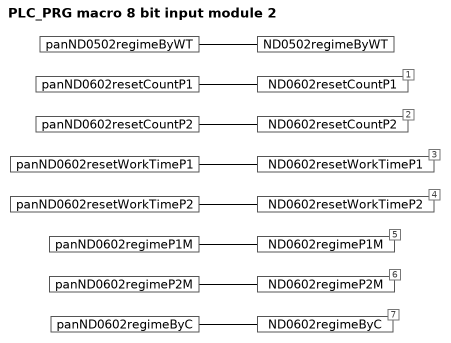
[picture p72: PLC_PRG macro 8 bit input module 2 (CFC)]
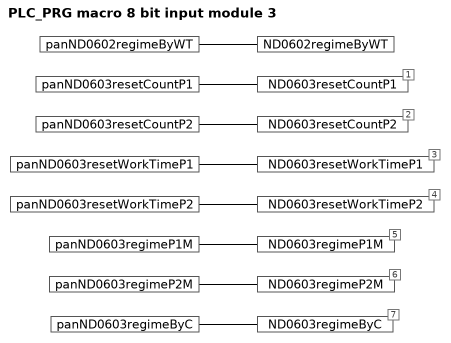
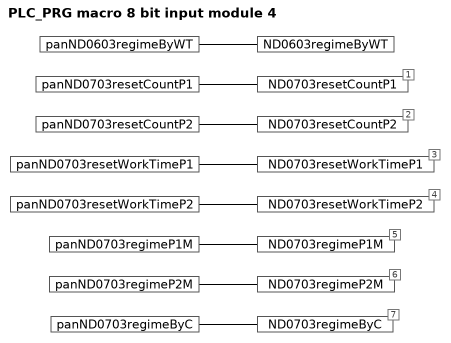
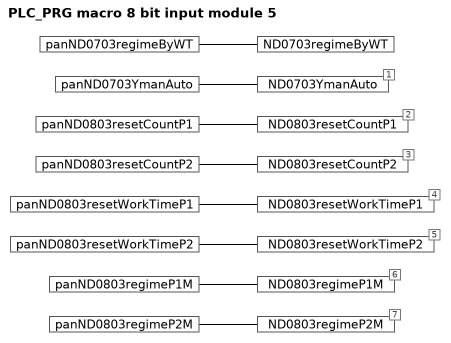
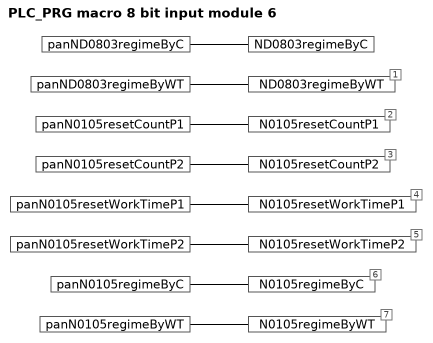
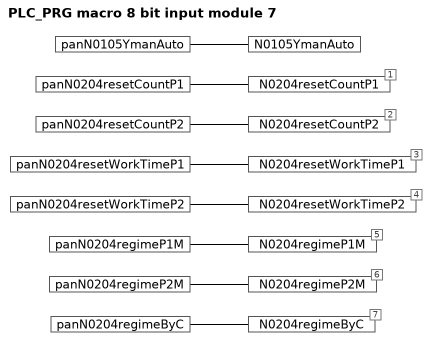
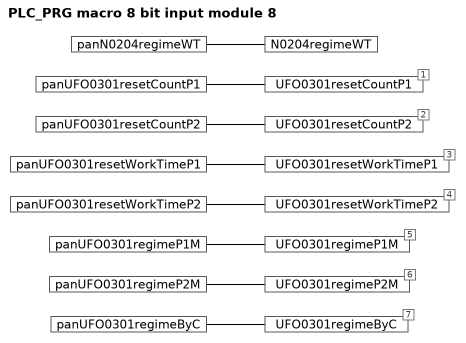
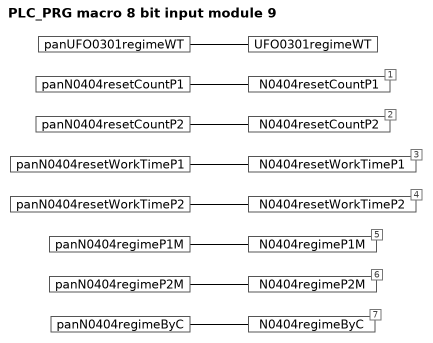
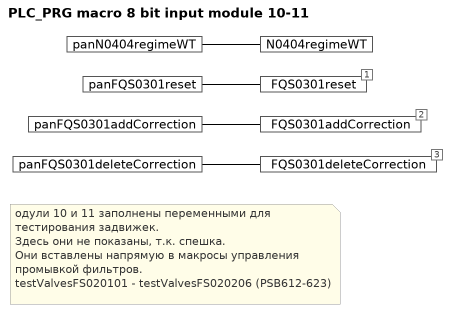
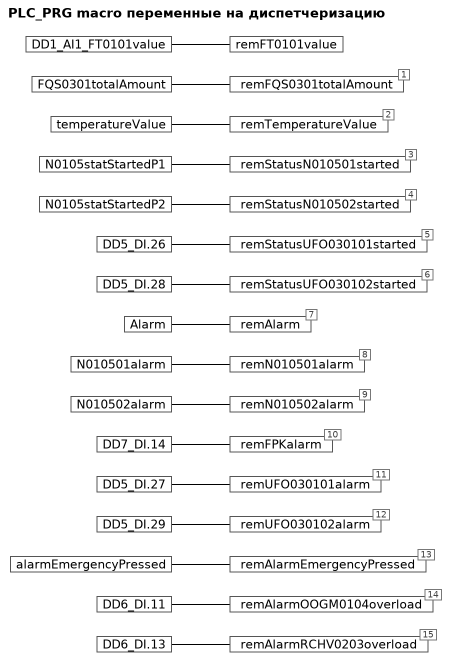
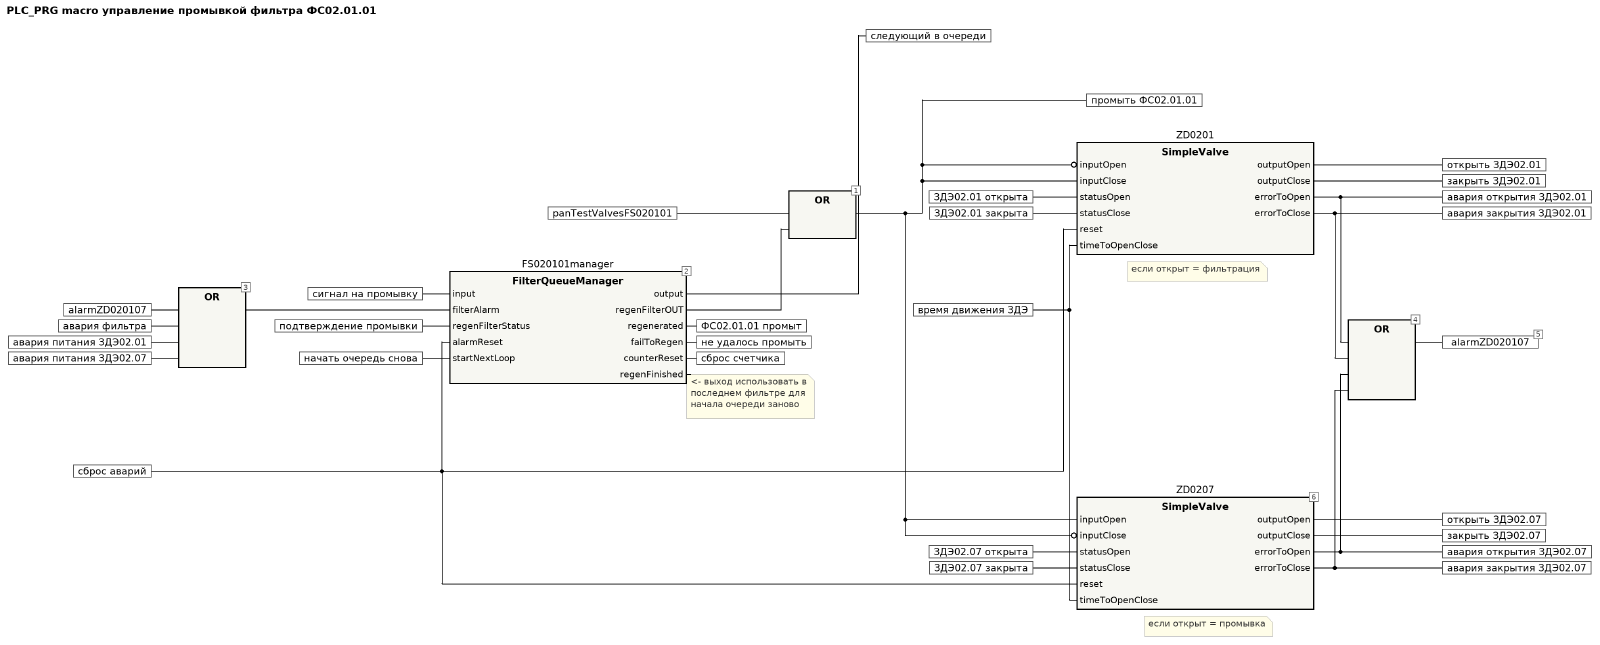
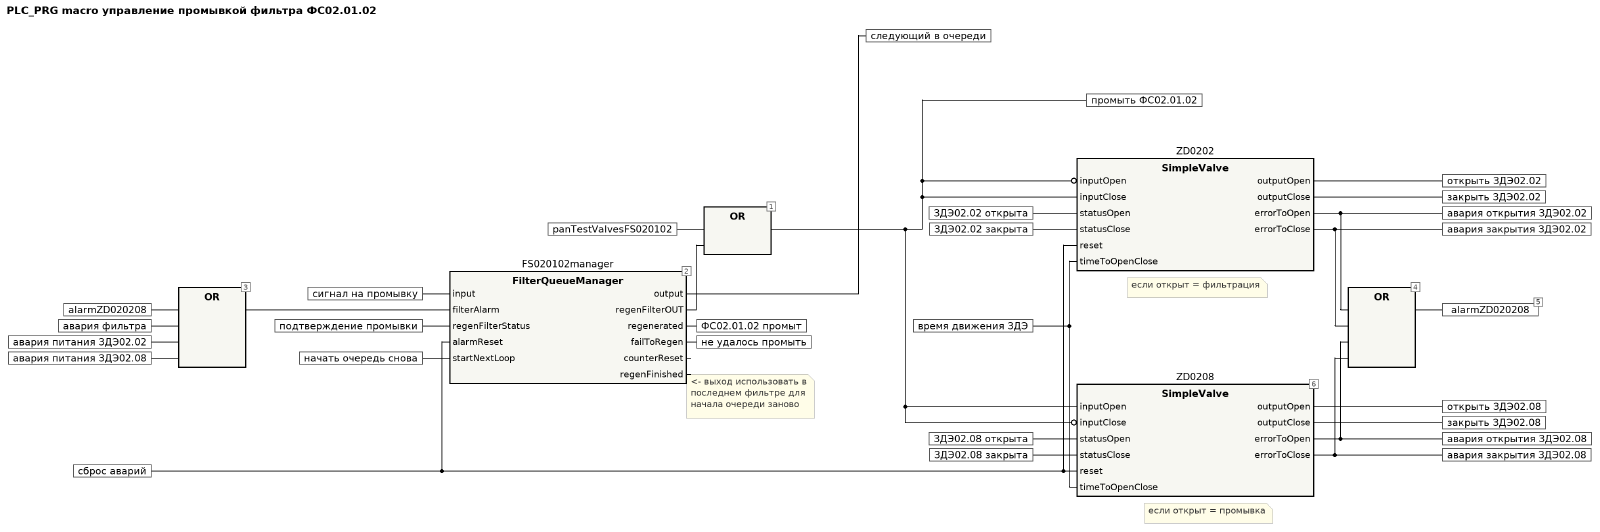
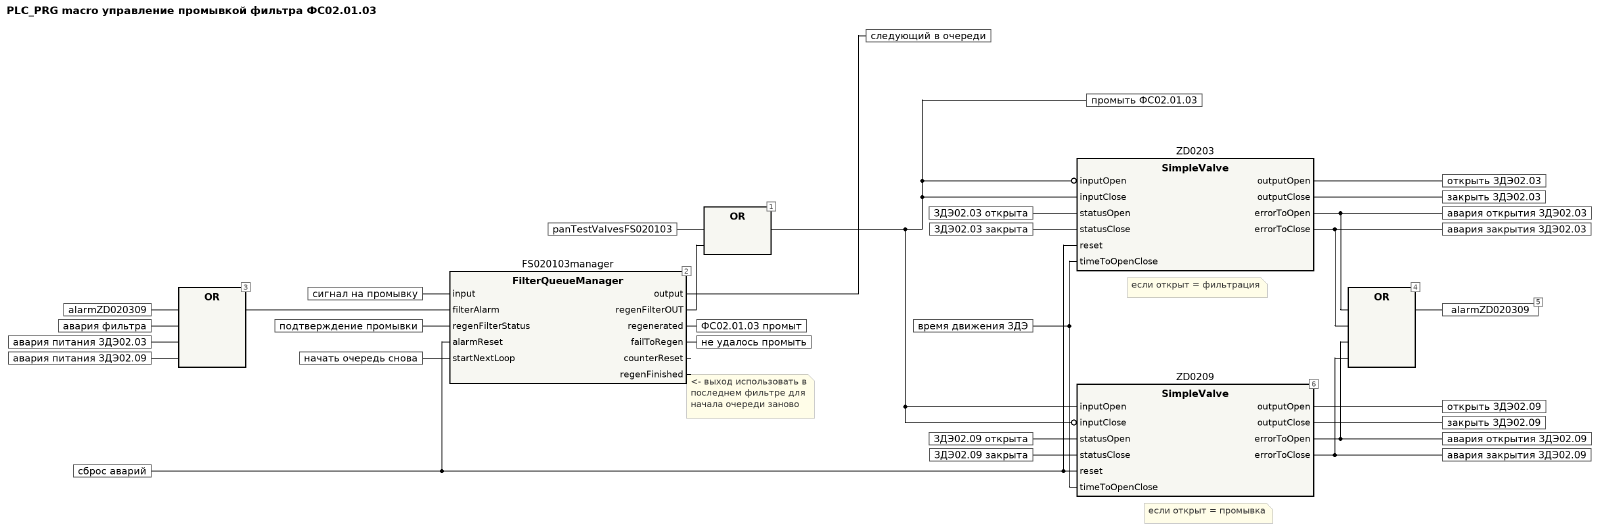
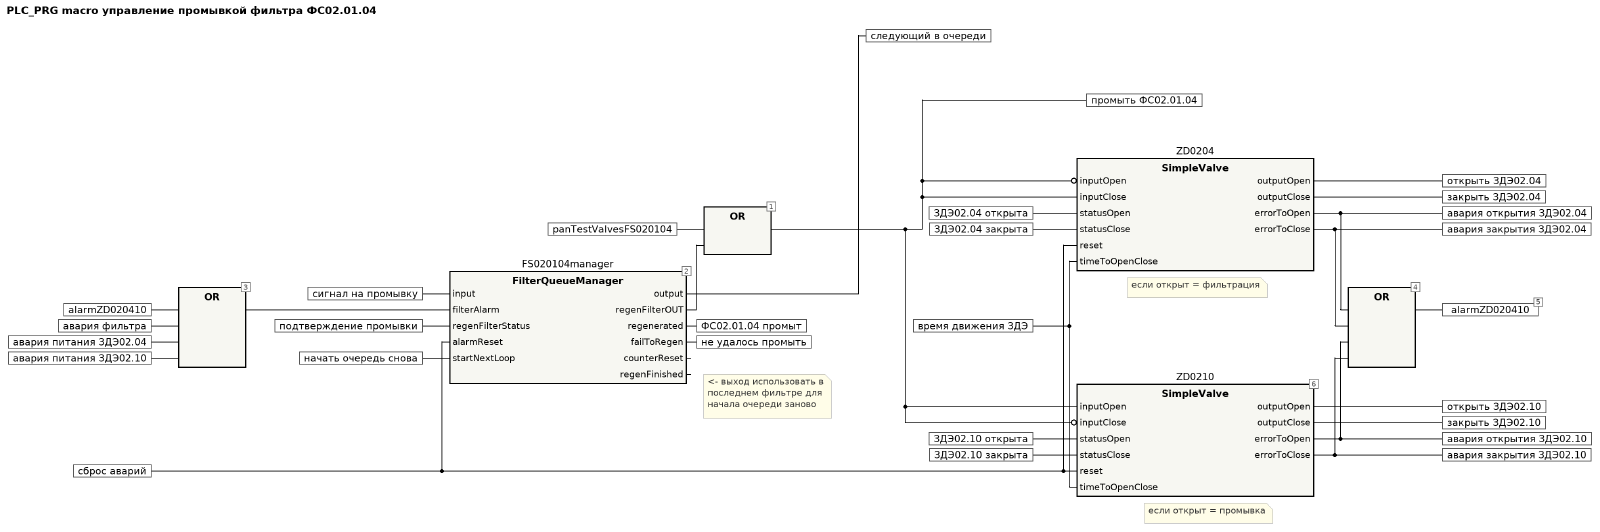
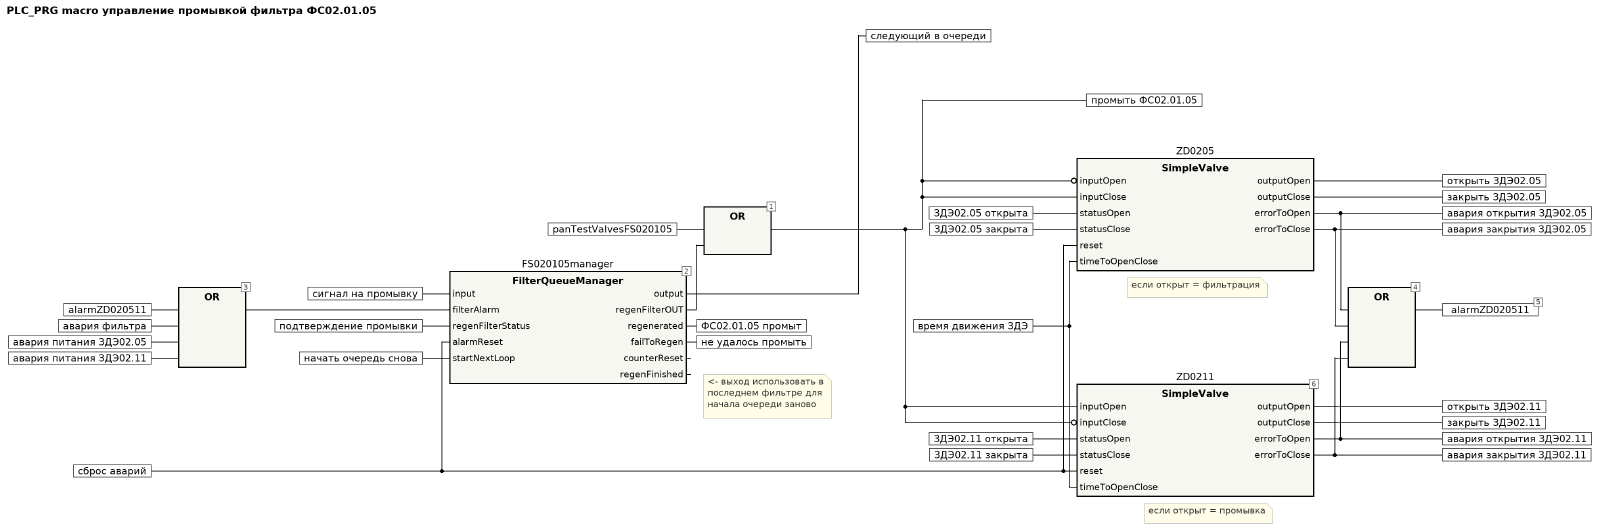
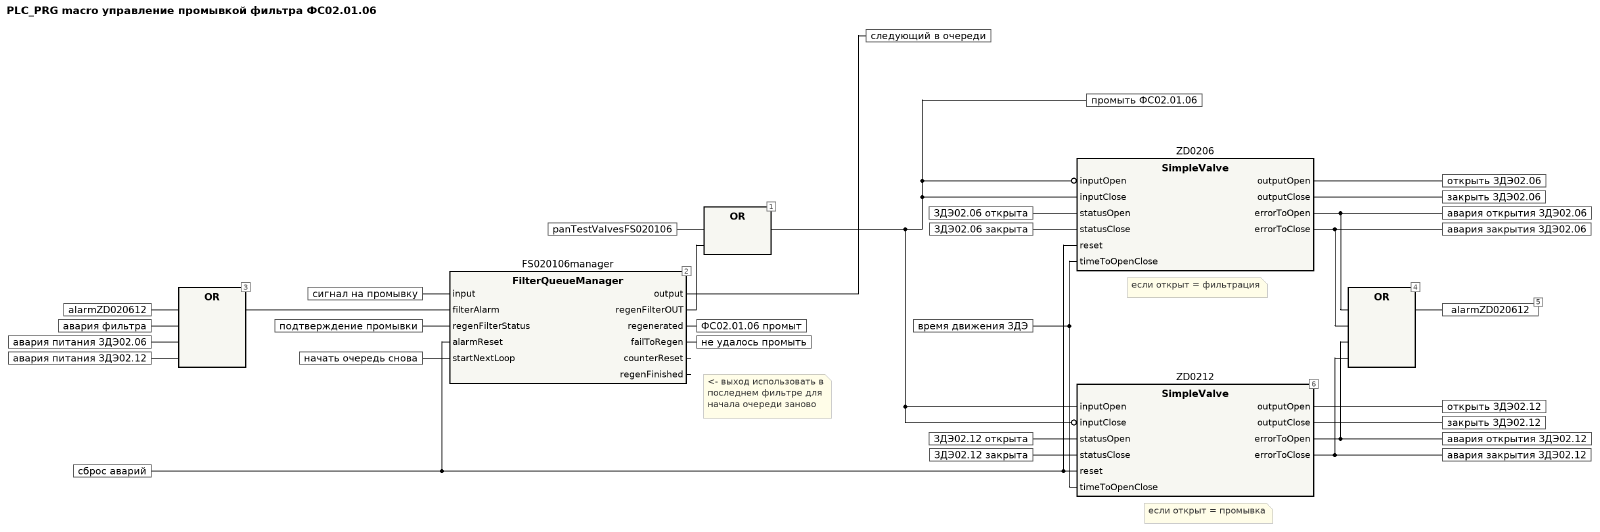
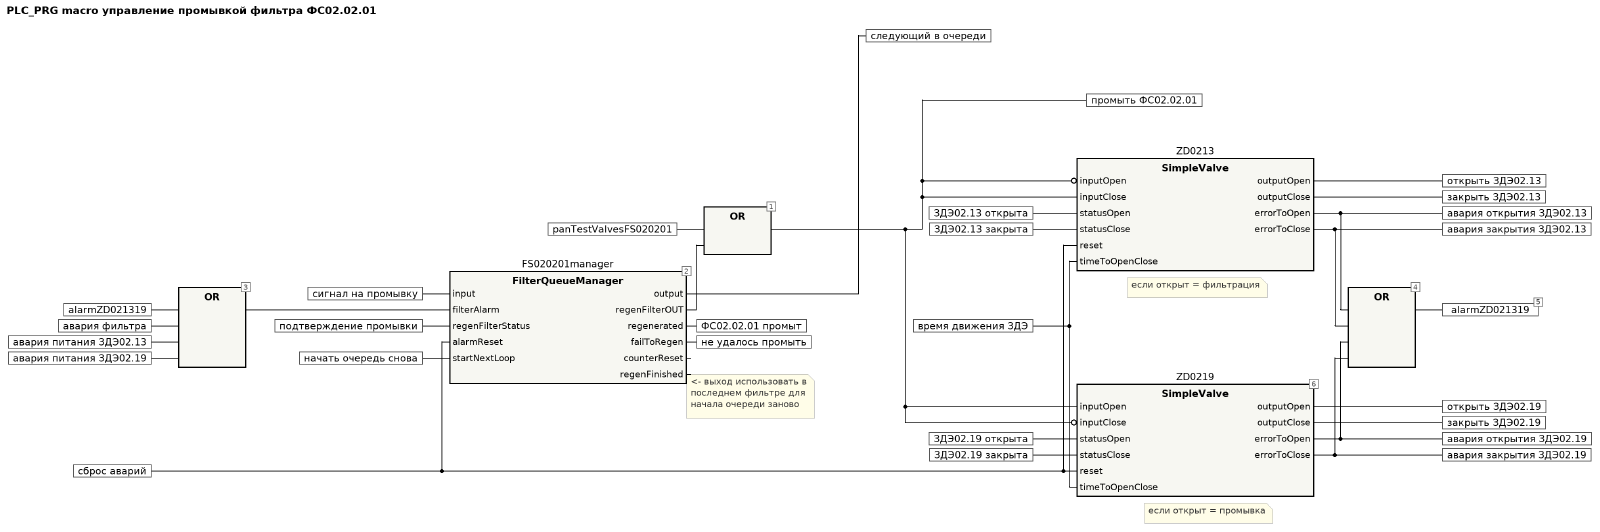
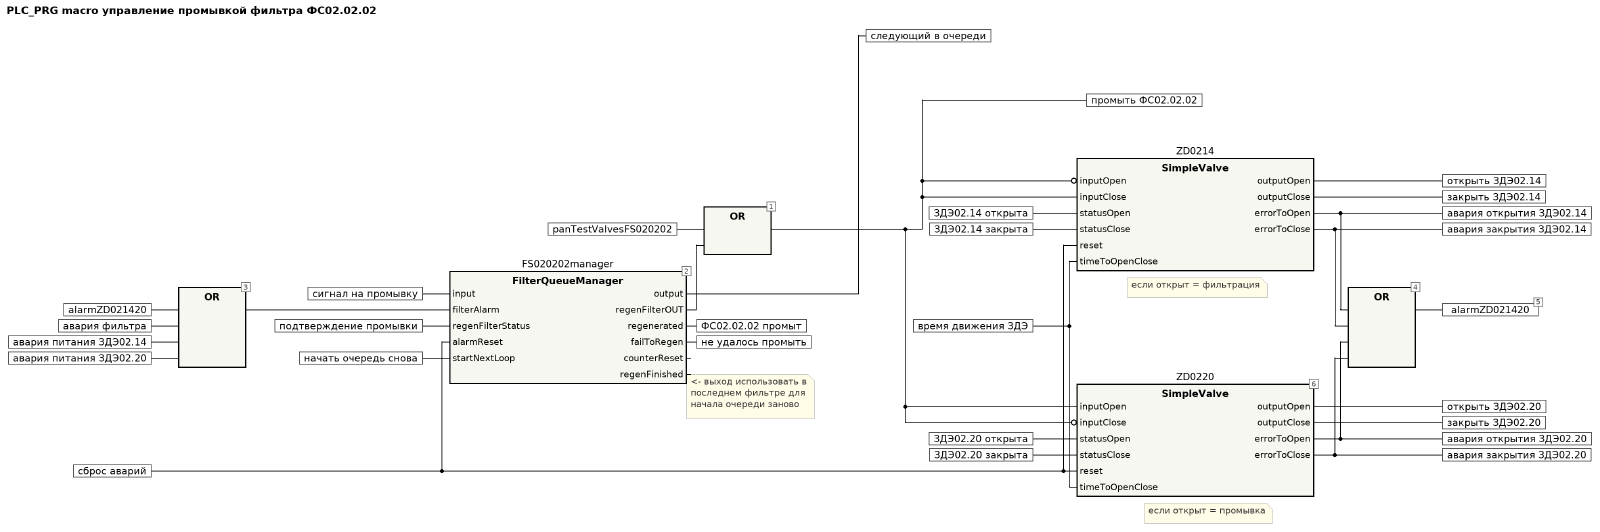
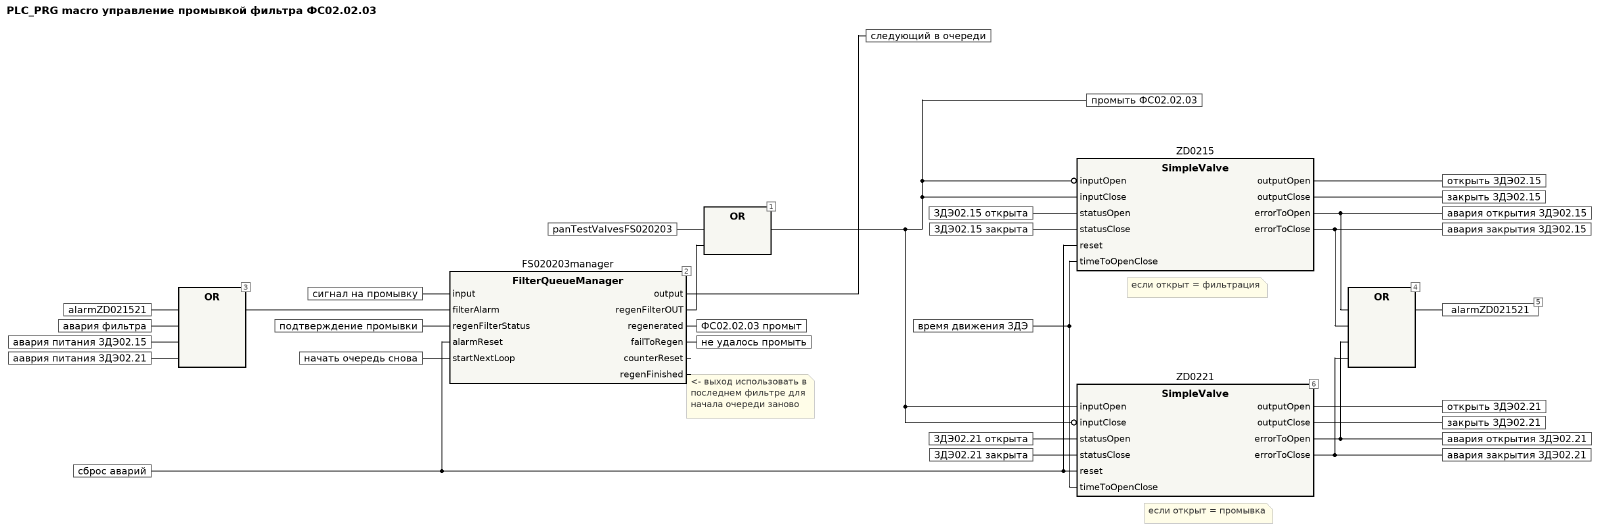
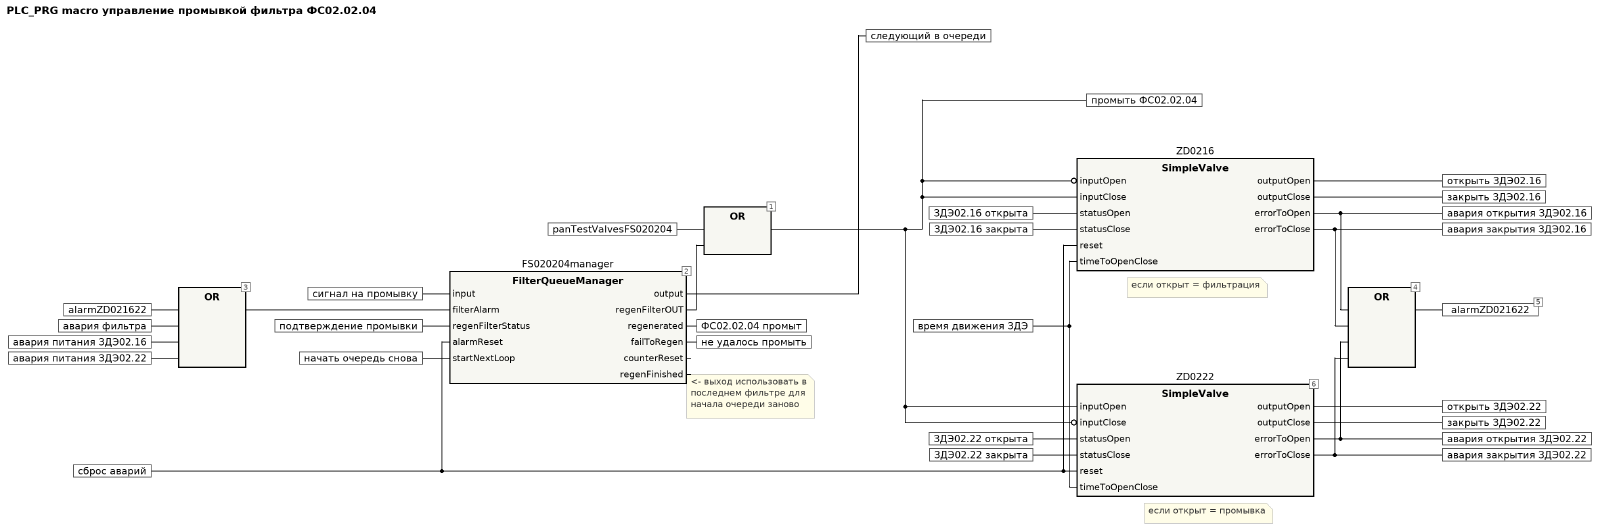
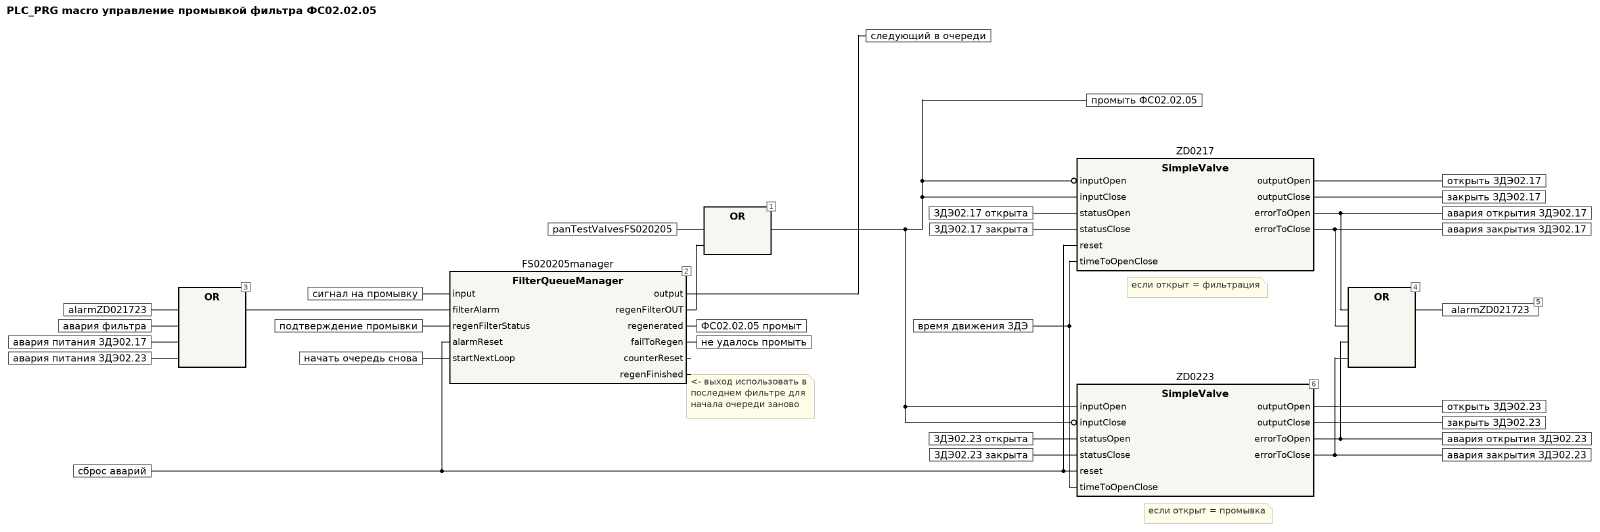
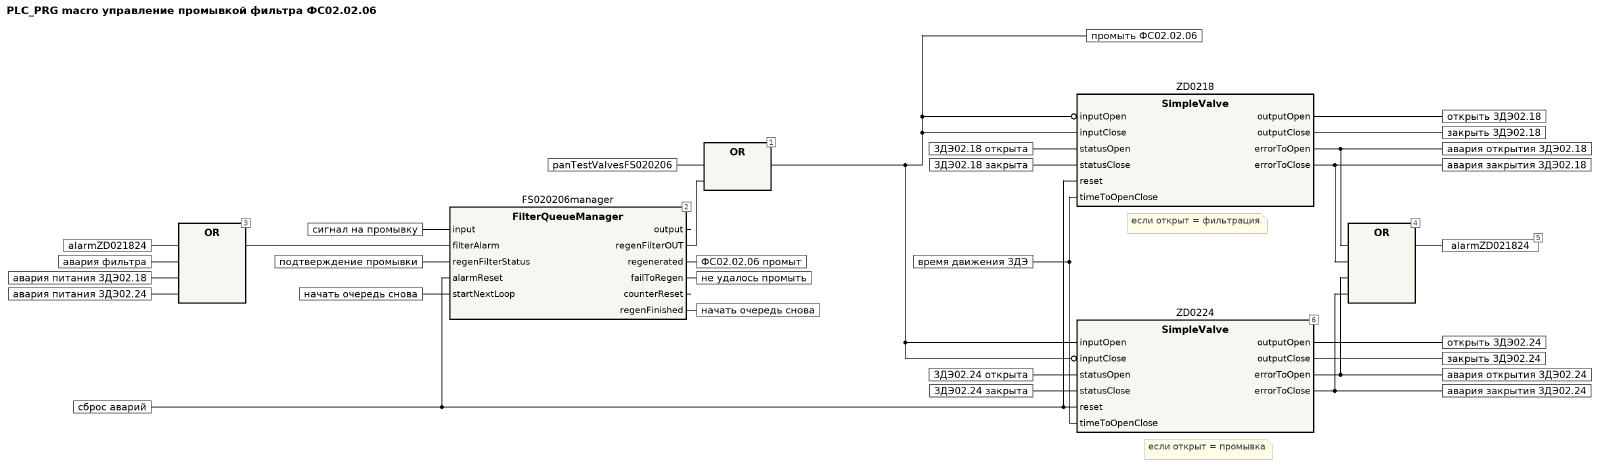
_CFC_ (* Continuous Function Chart, elements in execution order *)
(* 0 = перелив *)
(* авария обоих УФО, если проблемы / открытия/закрытия на одной из задвижек *)
(* авария питания ЗДЭ03.02 *)
(* авария питания ЗДЭ03.01 *)
(* статус-пуск Н01.05/02 *)
(* вкл КМ3 *)
(* Статус ПУСК / ЧРП Н01.05 *)
(* статус-пуск Н01.05/01 *)
(* вкл КМ2 *)
(* контроль обрыва или ошибок модулей в сети ПЛК *)
(* LSA01.02 перелив ОГМ01.04 *)
(* Нажат аварийный стоп. *)
(* авария сети (РКФ) *)
(* разрешение работы КНС / 1 = разрешено *)
(* Нажат аварийный стоп. *)
(* Блок управления разрешением работы КНС *)
(* авария сети (РКФ) *)
(* Авария питания клапанов КЭМ. *)
(* Авария питания розеток / управл.клапанов фильтров. *)
(* авария КНС *)
(* блок подачи сигнала на промывку *)
(* суммируем каждую секунду значение / мгновенного расхода в кубометрах в секунду *)
(* преобразуем расход из / кубометров в час в / кубометры в секунду *)
(* если есть расход / (больше нуля) *)
(* выдает импульс / каждую секунду *)
(* здесь мгновенный расход / в кубометрах в час (FT01.02) *)
(* Авария Н02.04/01 (0=авария) *)
(* Авария Н02.04/02 (0=авария) *)
(* промывка ФС02.01/06 *)
(* промывка ФС02.01/05 *)
(* промывка ФС02.01/04 *)
(* промывка ФС02.01/03 *)
(* промывка ФС02.01/02 *)
(* промывка ФС02.01/01 *)
(* пуск/стоп НД08.03/01 *)
(* пуск/стоп НД08.03/02 *)
(* пуск/стоп НД06.03/01 *)
(* пуск/стоп НД06.03/02 *)
(* пуск/стоп НД06.02/01 *)
(* пуск/стоп НД06.02/02 *)
(* пуск/стоп НД08.04 *)
(* пуск/стоп НД07.03/01 *)
(* пуск/стоп НД07.03/02 *)
(* авария М08.02 (УПФ) *)
(* авария М07.02 (УПЩ) *)
(* авария М06.04 (УПК) *)
(* работа М08.02 (УПФ) *)
(* работа М07.02 (УПЩ) *)
(* работа М06.04 (УПК) *)
(* Контроль, если УФО включили вручную, / а потока при этом нет. *)
(* авария УФО03.01/02 *)
(* работа УФО03.01/02 *)
(* авария УФО03.01/01 *)
(* Для подачи предостережения на пульте / оператора (при необходимости), а также / сигнализации лампой АВАРИЯ. *)
(* работа УФО03.01/01 *)
(* авария УФО03.01/02 *)
(* авария УФО03.01/01 *)
(* авария Н04.04/01 *)
(* авария Н04.04/02 *)
(* время контроля старта ФПК (по умолч.=3мин) *)
(* время работы ФПК после спада сигнала датч.осадка *)
(* запуск фильтрации *)
(* Защита от сухого хода насоса ФПК *)
(* датчик уровня осадка *)
(* Давление на входе ФПК (0...16 бар) *)
(* авария ФПК *)
(* подающий насос ФПК работает *)
(* ФПК готов к приему *)
(* ФПК не запустился *)
(* рН-метр QE01.02 на входе, / диапазон 0...14 *)
(* авария входа рН-метра QE01.01 *)
(* авария входа расходомера FT01.02 *)
(* расходомер FT01.01 на входе, / диапазон 0...600куб/час *)
(* авария НД08.04 *)
(* управление 4...20мА НД08.03/01 *)
(* пуск/стоп НД08.03/01 *)
(* пуск/стоп НД08.03/02 *)
(* управление 4...20мА НД08.03/02 *)
(* авария привода НД08.03/01 *)
(* авария привода НД08.03/02 *)
(* авария НД07.03/01 *)
(* авария НД07.03/02 *)
(* управление 4...20мА НД07.03/01 *)
(* управление 4...20мА НД07.03/02 *)
(* пуск/стоп НД07.03/01 *)
(* пуск/стоп НД07.03/02 *)
(* авария НД07.03/01 *)
(* авария НД07.03/02 *)
(* авария НД06.03/01 *)
(* авария НД06.03/02 *)
(* авария НД06.02/01 *)
(* авария НД06.02/02 *)
(* управление 4...20мА НД06.03/01 *)
(* пуск/стоп НД06.03/01 *)
(* пуск/стоп НД06.03/02 *)
(* управление 4...20мА НД06.03/02 *)
(* авария НД06.03/01 *)
(* авария НД06.03/02 *)
(* управление 4...20мА НД06.02/01 *)
(* пуск/стоп НД06.02/01 *)
(* пуск/стоп НД06.02/02 *)
(* управление 4...20мА НД06.02/02 *)
(* авария НД06.02/01 *)
(* авария НД06.02/02 *)
(* ошибка блока дозирования НД05.02 *)
(* авария входа датчика температуры *)
(* лампа АВАРИЯ *)
(* датчик температуры в помещении / (метран) диапазон: 0...+100С *)
(* управление 4...20мА НД05.02/01 *)
(* пуск/стоп НД05.02/01 *)
(* авария НД05.02/01 *)
(* авария НД05.02/02 *)
(* пуск/стоп НД05.02/02 *)
(* управление 4...20мА НД05.02/02 *)
(* АВАРИИ *)
(* авария привода НД08.03/01 *)
(* авария привода НД08.03/02 *)
(* авария НД08.04 *)
(* насос Н04.01 работает *)
(* пуск/стоп НД08.04 *)
(* управление 4...20мА НД08.04 *)
(* авария входа расходомера FT01.01 *)
(* расходомер FT01.02 на входе, / диапазон 0...600куб/час *)
(* рН-метр QE01.01 на входе, / диапазон 0...14 *)
(* авария входа рН-метра QE01.02 *)
(* сухой ход НД08.03/01 *)
(* сухой ход НД08.03/02 *)
(* сухой ход НД08.03/01 *)
(* сухой ход НД08.03/02 *)
(* LSA01.02 перелив ОГМ01.04 *)
(* Инициализирует требуемые булевые переменные / в момент старта выполнения программы. *)
(* Статус ПУСК ЧРП Н01.05 *)
(* LS01.03 - рабочий верхний уровень ОГМ01.04 автоматический пуск 01.05 *)
(* LS01.04 - нижний уровень ОГМ01.04, сухой ход Н01.05 *)
(* SA1 Ручной выбор Н01.05/01 = главный *)
(* SA1 Ручной выбор Н01.05/02 = главный *)
(* Стоп  Н01.05 (сброс самоподхвата реле) *)
(* время на создание потока *)
(* Пуск  Н01.05 *)
(* КМ1 питание ЧРП *)
(* КМ2 питание насоса 1 *)
(* КМ3 питание насоса 2 *)
(* Авария ЧРП Н01.05 *)
(* термоконтакт Н01.05/01 *)
(* термоконтакт Н01.05/02 *)
(* авария питания ЗДЭ02.25 *)
(* LSА02.01 Перелив РЧВ02.03 *)
(* Давление на входе ФПК / 0...16 бар (мах допуст.10) *)
(* Авария входа AI6 ПЛК, давл.ФПК *)
(* авария ФПК *)
(* Открыть КШЭ04.01 *)
(* статус КШЭ04.01 открыт *)
(* Закрыть КШЭ04.01 *)
(* статус КШЭ04.01 закрыт *)
(* подающий насос ФПК работает *)
(* стоп Н04.04 *)
(* пуск Н04.04/02 *)
(* пуск Н04.04/01 *)
(* авт.пуск Н04.04 *)
(* сухой ход Н04.04, 0=защита *)
(* авария Н04.04/01, 0=авария *)
(* авария Н04.04/02, 0=авария *)
(* импульсный расходомер *)
(* Авария Н02.04/01 (0=авария) *)
(* Авария Н02.04/02 (0=авария) *)
(* промывка ФС02.02/06 *)
(* промывка ФС02.02/05 *)
(* промывка ФС02.02/04 *)
(* промывка ФС02.02/03 *)
(* промывка ФС02.02/02 *)
(* промывка ФС02.02/01 *)
(* Клапан КЭМ05.01 открыт. *)
(* Клапан КЭМ06.01 открыт. *)
(* Клапан КЭМ07.01 открыт. *)
(* Клапан КЭМ08.01 открыт. *)
(* Сухой ход Н02.04 (LS02.03) 0=сух.ход *)
(* Стоп Н02.04 *)
(* Пуск Н02.04/01 *)
(* Пуск Н02.04/02 *)
(* текущий объем *)
(* заданный до промывки объем *)
(* 0=авария *)
(* авария (при 0) ФС02.01/06 *)
(* авария (при 0) ФС02.01/05 *)
(* авария (при 0) ФС02.01/04 *)
(* авария (при 0) ФС02.01/03 *)
(* авария (при 0) ФС02.01/02 *)
(* авария (при 0) ФС02.01/01 *)
(* авария (при 0) ФС02.02/06 *)
(* авария (при 0) ФС02.02/05 *)
(* авария (при 0) ФС02.02/04 *)
(* авария (при 0) ФС02.02/03 *)
(* авария (при 0) ФС02.02/02 *)
(* авария (при 0) ФС02.02/01 *)
(* сброс счетчика стоков до следующей промывки *)
(* подсчет общего объема стоков, прошедшего через расходомер FT01.02 *)
(* очередь передается на 2 ступень *)
(* авария питания ЗДЭ02.01 *)
(* авария питания ЗДЭ02.02 *)
(* авария питания ЗДЭ02.03 *)
(* авария питания ЗДЭ02.04 *)
(* авария питания ЗДЭ02.05 *)
(* авария питания ЗДЭ02.06 *)
(* авария питания ЗДЭ02.07 *)
(* авария питания ЗДЭ02.08 *)
(* авария питания ЗДЭ02.09 *)
(* авария питания ЗДЭ02.10 *)
(* авария питания ЗДЭ02.11 *)
(* авария питания ЗДЭ02.12 *)
(* авария питания ЗДЭ02.13 *)
(* авария питания ЗДЭ02.14 *)
(* авария питания ЗДЭ02.15 *)
(* авария питания ЗДЭ02.16 *)
(* авария питания ЗДЭ02.17 *)
(* авария питания ЗДЭ02.18 *)
(* авария питания ЗДЭ02.19 *)
(* авария питания ЗДЭ02.20 *)
(* авария питания ЗДЭ02.21 *)
(* авария питания ЗДЭ02.22 *)
(* авария питания ЗДЭ02.23 *)
(* авария питания ЗДЭ02.24 *)
(* инвертирование сигнала, чтобы все аварии / обозначались как 1 (TRUE) *)
(* авария НД05.02/01 *)
(* авария НД05.02/02 *)
(* авария питания КШЭ04.01 *)
(* 1=открыть; 0 = закрыть *)
(* в этом макросе лежит управление режимом тестирования задвижек ЗДЭ03 / Тестирование запрещает автоматический запуск УФО от ПЛК *)
#0 rTrigStartInitializer:R_TRIG(CLK: TRUE)
#1 startInitializer <= #0.Q
#2 MACRO контроль температуры в помещении(pin 1 "вход датчика температуры": DD1_AI0, pin 2 "минимально допустимая температура в помещении": maxTemperature, pin 3 "максимально допустимая температура в помещении": minTemperature)
	(* задаем границы допустимой температуры в помещении / проверяем что измеренное значение в заданном диапазоне *)
	(* не смотрим конкретный тип ошибки / (работает не точно, обрыв определяет как слишком маленькое значение) / если не равно 0 - значит на входе ошибка *)
	#3 DD1_AI0_temperature:DECODE_FLOAT(VALUE: pin 1, DEF_VALUE: -)
	#4 NE(#3._ERR, 0)
	out 2 "авария датчика температуры" <= #4
	out 1 "температура в помещении" <= #3.OUT_VALUE
	#5 REAL_TO_INT(#3.OUT_VALUE)
	#6 temperatureLimits:LIMITALARM(IN: #5, HIGH: pin 3, LOW: pin 2)
	out 3 "температура выше заданного диапазона" <= #6.O
	out 4 "температура ниже заданного диапазона" <= #6.U
	#7 temperatureLimits:LIMITALARM(IN: -, HIGH: -, LOW: -)
END_MACRO
#8 temperatureValue <= #2.out 1
#9 DD1_AI0_error <= #2.out 2
#10 alarmHighTemperature <= #2.out 3
#11 alarmLowTemperature <= #2.out 4
#12 OR(testKSHE0401, DD7_DI.13)
#13 MACRO клапан шаровый перед ФПК (КШЭ04.01)(pin 1 "сигнал "подающий насос ФПК" работает": #12, pin 2 "статус КШЭ04.01 открыт": DD9_DI.2, pin 3 "статус КШЭ04.01 закрыт": DD9_DI.3, pin 4 "сброс аварий": alarmReset, pin 5 "время на открытие/закрытие": timeToOpenCloseValve)
	#14 FPKkshe0401DelayToOpen:TON(IN: #16.outputOpen, PT: T#1s)
	out 1 "выход на открытие КШЭ04.01" <= #14.Q
	#15 FPKkshe0401DelayToClose:TON(IN: #16.outputClose, PT: T#1s)
	out 2 "выход на закрытие КШЭ04.01" <= #15.Q
	#16 FPKkshe0401:SimpleValve(inputOpen: pin 1, inputClose: #17, statusOpen: pin 2, statusClose: pin 3, reset: pin 4, timeToOpenClose: pin 5)
	#17 NOT(pin 1)
	out 3 "авария на открытие КШЭ04.01" <= #16.errorToOpen
	out 4 "авария на закрытие КШЭ04.01" <= #16.errorToClose
END_MACRO
#18 DD4_DO.2 <= #13.out 1
#19 DD4_DO.3 <= #13.out 2
#20 FPKkshe0401errorToOpen <= #13.out 3
#21 FPKkshe0401errorToClose <= #13.out 4
#22 OR(DD1_AI0_error, DD1_AI1_error, DD1_AI2_error, DD1_AI3_error, DD1_AI4_error, alarmHighTemperature, alarmLowTemperature, ND0502dosingError, ND0602dosingError, ND0603dosingError, ND0803dosingError, ND0804dosingError, DD1_DI6, DD1_DI7, N010501alarm, N010502alarm, ZDE0225errorToOpen, ZDE0225errorToClose, DD7_DI.14, FPKnotStarted, DD1_AI5_error, FPKkshe0401errorToOpen, FPKkshe0401errorToClose, DD5_DI.27, DD5_DI.29, filterFailToRegen020101, errorToOpenZD0201, errorToCloseZD0201, errorToOpenZD0207, errorToCloseZD0207, filterFailToRegen020102, errorToOpenZD0202, errorToCloseZD0202, errorToOpenZD0208, errorToCloseZD0208, filterFailToRegen020103, errorToOpenZD0203, errorToCloseZD0203, errorToOpenZD0209, errorToCloseZD0209, filterFailToRegen020104, errorToOpenZD0204, errorToCloseZD0204, errorToOpenZD0210, errorToCloseZD0210, filterFailToRegen020105, errorToOpenZD0205, errorToCloseZD0205, errorToOpenZD0211, errorToCloseZD0211, filterFailToRegen020106, errorToOpenZD0206, errorToCloseZD0206, errorToOpenZD0212, errorToCloseZD0212, filterFailToRegen020201, errorToOpenZD0213, errorToCloseZD0213, errorToOpenZD0219, errorToCloseZD0219, filterFailToRegen020202, errorToOpenZD0214, errorToCloseZD0214, errorToOpenZD0220, errorToCloseZD0220, filterFailToRegen020203, errorToOpenZD0215, errorToCloseZD0215, errorToOpenZD0221, errorToCloseZD0221, filterFailToRegen020204, errorToOpenZD0216, errorToCloseZD0216, errorToOpenZD0222, errorToCloseZD0222, filterFailToRegen020205, errorToOpenZD0217, errorToCloseZD0217, errorToOpenZD0223, errorToCloseZD0223, filterFailToRegen020206, errorToOpenZD0218, errorToCloseZD0218, errorToOpenZD0224, errorToCloseZD0224, alarmPLKnetwork, alarmND050201, alarmND050202, alarmND060201, alarmND060202, alarmND060301, alarmND060302, alarmND070301, alarmND070302, alarmND080301, alarmND080302, alarmND0804, alarmOGM0104overload, alarmRCHV0203overload, alarmN040402, alarmN040401, alarmM0604, alarmM0702, alarmM0802, alarmN020401, alarmN020402, alarmFS020101, alarmFS020102, alarmFS020103, alarmFS020104, alarmFS020105, alarmFS020106, alarmFS020201, alarmFS020202, alarmFS020203, alarmFS020204, alarmFS020205, alarmFS020206, alarmZDE0201power, alarmZDE0202power, alarmZDE0203power, alarmZDE0204power, alarmZDE0205power, alarmZDE0206power, alarmZDE0207power, alarmZDE0208power, alarmZDE0209power, alarmZDE0210power, alarmZDE0211power, alarmZDE0212power, alarmZDE0213power, alarmZDE0214power, alarmZDE0215power, alarmZDE0216power, alarmZDE0217power, alarmZDE0218power, alarmZDE0219power, alarmZDE0220power, alarmZDE0221power, alarmZDE0222power, alarmZDE0223power, alarmZDE0224power, alarmZDE0225power, alarmKSHE0401power, alarmKNS, alarmPowerSocketFS, alarmKEMvalvesPower, alarmEmergencyPressed, alarmRKF, errorToOpenZDE0301, errorToCloseZDE0301, errorToOpenZDE0302, errorToCloseZDE0302, alarmZDE0301power, alarmZDE0302power)
#23 DD1_DO11 <= #22
#24 alarm <= #22
#25 MACRO контроль аналогового входа DD1_AI1(pin 1 "вход": DD1_AI1)
	(* Не смотрим конкретную ошибку, / определяем,что вход неисправен без расшифровки. *)
	#26 DD1_AI1_FT0101:DECODE_FLOAT(VALUE: pin 1, DEF_VALUE: -)
	#27 NE(#26._ERR, 0)
	out 2 "авария" <= #27
	out 1 "выход" <= #26.OUT_VALUE
END_MACRO
#28 DD1_AI1_FT0101value <= #25.out 1
#29 DD1_AI1_error <= #25.out 2
#30 MACRO контроль аналогового входа DD1_AI2(pin 1 "вход": DD1_AI2)
	(* Не смотрим конкретную ошибку, / определяем,что вход неисправен без расшифровки. *)
	#31 DD1_AI2_FT0102:DECODE_FLOAT(VALUE: pin 1, DEF_VALUE: -)
	#32 NE(#31._ERR, 0)
	out 2 "авария" <= #32
	out 1 "выход" <= #31.OUT_VALUE
END_MACRO
#33 DD1_AI2_FT0102value <= #30.out 1
#34 DD1_AI2_error <= #30.out 2
#35 MACRO управление Н01.05 (поддержание заданного расхода по FT01.02)(pin 1 "статус ПУСК ЧРП (реле)": DD5_DI.4, pin 2 "LS01.03 раб.уров.": DD6_DI.12, pin 3 "LS01.04 ниж.уров.(сух.ход)": DD5_DI.0, pin 4 "SA1ручной выб.Н01.05/01-главный": DD5_DI.5, pin 5 "SA1ручной выб.Н01.05/02-главный": DD5_DI.6, pin 6 "включить режим "по кол.вкл."": N0105regimeByC, pin 7 "включить режим "по наработке"": N0105regimeByWT, pin 8 "значение расхода от FT01.02": DD1_AI2_FT0102value, pin 9 "уставка расхода": N0105flowSetValue, pin 10 "время на создание потока": N0105minFlowTime, pin 11 "Р-коэфф.": N0105koeffP, pin 12 "I-коэфф": N0105koeffI, pin 13 "Д-коэфф": N0105koeffD, pin 14 "управление ЧРП в ручн.реж.(4...20мА)": N0105YoutManual, pin 15 "переключатель управление ЧРП РУЧН/АВТ": N0105YmanAuto, pin 16 "мин.допустимый расход": N0105minFlow, pin 17 "термоконтакт Н01.05/01": DD5_DI.2, pin 18 "термоконтакт Н01.05/02": DD5_DI.3, pin 19 "авария ЧРП Н01.05": DD5_DI.1, pin 20 "сброс аварии": alarmReset, pin 21 "сброс кол-ва вкл.Н01.05/01": N0105resetCountP1, pin 22 "сброс кол-ва вкл.Н01.05/02": N0105resetCountP2, pin 23 "сброс наработки Н01.05/01": N0105resetWorkTimeP1, pin 24 "сброс наработки Н01.05/02": N0105resetWorkTimeP2)
	(* время на создание потока *)
	(* Пуск  Н01.05 *)
	(* режимы по количеству включений,  или по наработке / активны если оба входа SA1 не активны *)
	(* управление Н01.05 - поддержание / заданного расхода по FT01.02 *)
	(* по умолчанию при старте программы *)
	(* если на входе true / то нижнее значение, / иначе то, что посередине *)
	(* Если насос создает давление меньше / указанного, то авария. *)
	#36 OR(pin 2, #37.Q)
	#37 N0105startTrig:R_TRIG(CLK: pin 1)
	#38 N0105stopTrig:F_TRIG(CLK: pin 1)
	#39 N0105startTrigg:RS(SET: #36, RESET1: #41)
	#40 N0105regime:choosePumpRegime(start: #39.Q1, pump1Main: pin 4, pump2Main: pin 5, byCounter: #44, byWorkTime: #50)
	out 2 "статус режим "Н01.05/01 - главный"" <= #40.pump1MainActive
	out 3 "статус режим "Н01.05/02 - главный"" <= #40.pump2MainActive
	out 4 "статус режим "по кол-ву вкл."" <= #40.byCounterActive
	#41 OR(#38.Q, #42)
	out 5 "статус режим "по наработке"." <= #40.byWorkTimeActive
	#42 NOT(pin 3)
	#43 NOT(#39.Q1)
	out 1 "СТОП (сброс самоподхвата реле пуска ЧРП)." <= #43
	#44 AND(NOT pin 4, NOT pin 5, #47.Q1)
	#45 OR(pin 6, startInitializer)
	#46 N0105regByCinit:R_TRIG(CLK: #45)
	#47 N0105regByCtrig:RS(SET: #46.Q, RESET1: #55.Q)
	#48 N0105twoPumpOneDriveManager:TwoPumpOneDriveManager(startStopPump1: #40.startPump1, startStopPump2: #40.startPump2, alarmPump1: N010501alarm, alarmPump2: N010502alarm, alarmReset: alarmReset, counterStart: #40.startByCounter, Pump1ResetCounter: pin 21, Pump2ResetCounter: pin 22, ValueToResetCounter: -, workTimeStart: #40.startByWorkTime, workTimePump1Reset: pin 23, workTimePump2Reset: pin 24, timeKM1off: -, timeKM23DelayON: -, timeKM23offDelay: -, timeReadyToStartDelay: -)
	out 6 "кол-во включений Н01.05/01" <= #48.counterPump1
	#49 AND(#48.pump1active, #65)
	out 7 "кол-во включений Н01.05/02" <= #48.counterPump2
	out 8 "наработка Н01.05/01" <= #48.currentWorkTimePump1
	out 15 "авария Н01.05/01" <= #53.Q1
	#50 AND(NOT pin 4, NOT pin 5, #56.Q1)
	out 9 "наработка Н01.05/02" <= #48.currentWorkTimePump2
	out 10 "КМ1-питание ЧРП" <= #48.DriveKM
	#51 AND(#48.pump1active, #57)
	#52 OR(#49, #51)
	#53 N010501alarmTrig:RS(SET: #52, RESET1: pin 20)
	#54 N010501alarm <= #53.Q1
	#55 N0105regWTinit:R_TRIG(CLK: pin 7)
	#56 N0105regWTtrig:RS(SET: #55.Q, RESET1: #46.Q)
	out 11 "КМ2-питание Н01.05/01" <= #48.pump1KM
	out 12 "КМ3-питание Н01.05/02" <= #48.pump2KM
	#57 OR(NOT pin 17, NOT pin 19)
	out 13 "пуск ЧРП (Н01.05)" <= #48.driveStart
	#58 OR(NOT pin 19, NOT pin 18)
	out 16 "авария Н01.05/02" <= #61.Q1
	#59 AND(#58, #48.pump2active)
	#60 OR(#59, #63)
	#61 N010502alarmTrig:RS(SET: #60, RESET1: pin 20)
	#62 N010502alarm <= #61.Q1
	#63 AND(#48.pump2active, #65)
	#64 N0105timerminFlow:TON(IN: #48.driveStart, PT: pin 10)
	#65 AND(#64.Q, #66)
	#66 LE(pin 8, pin 16)
	#67 SEL(#48.driveStart, 0, #68.Y)
	out 14 "управление ЧРП (4...20мА)" <= #67
	#68 N0105pidReg:PID(ACTUAL: pin 8, SET_POINT: pin 9, KP: pin 11, TN: pin 12, TV: pin 13, Y_MANUAL: pin 14, Y_OFFSET: -, Y_MIN: 4, Y_MAX: 20, MANUAL: pin 15, RESET: #68.OVERFLOW)
END_MACRO
#69 DD4_DO.13 <= #35.out 1
#70 N0105statRegimeP1M <= #35.out 2
#71 N0105statRegimeP2M <= #35.out 3
#72 N0105statRegimeByC <= #35.out 4
#73 N0105statRegimeByWT <= #35.out 5
#74 N0105counterP1 <= #35.out 6
#75 N0105counterP2 <= #35.out 7
#76 N0105workTimeP1 <= #35.out 8
#77 N0105workTimeP2 <= #35.out 9
#78 DD2_DO.0 <= #35.out 10
#79 DD2_DO.1 <= #35.out 11
#80 DD2_DO.2 <= #35.out 12
#81 DD1_DO0 <= #35.out 13
#82 DD1_AO0 <= #35.out 14
#83 N010501alarm <= #35.out 15
#84 N010502alarm <= #35.out 16
#85 MACRO Сигналы работы с ФП04.02 (фильтр-пресс)(pin 1 "датчик уровня осадка": DD7_DI.15, pin 2 "время работы ФПК (после выкл.датч.осадка)": FPKtimeToWork, pin 3 "защита от сухого хода": DD6_DI.10, pin 4 "ошибка входа AI (обрыв)": DD1_AI5_error, pin 5 "авария ФПК": DD7_DI.14, pin 6 "фильтр-пресс готов к приему": DD7_DI.12, pin 7 "давление на входе в ФПК": DD1_AI5_FPKpressureValue, pin 8 "мах допустимое давление": FPKmaxPressureValue, pin 9 "подающий насос ФПК работает": DD7_DI.13, pin 10 "время контроля старта ФПК": FPKnotStartedTime, pin 11 "сброс аварий": alarmReset)
	(* ФПК готов к приему осадка *)
	(* LS01.01-нижн.уровень на входе ОГМ01.04 / защита от сух. хода насоса ФПК *)
	(* LES01.01-сигнал датчика уровня осадка ОГМ01.04 / запуск процесса фильтрации *)
	(* Время работы ФПК после / спада сигнала уровня осадка / по умолч.15мин. *)
	(* Давление на входе ФПК / 0...16 бар (мах допуст.10) *)
	(* максимально допустимое давление / на входе ФПК *)
	(* Условие сброса сигнала о грязном фильтр-прессе: / 1. Пропал сигнал о готовности ФПК; / 2. Появился сигнал о готовности ФПК. / Это значит, что оператор раздвигал плиты, / чистил и снова сдвигал их. *)
	#86 FPKneedToCleanResetFtrig:F_TRIG(CLK: FPKneedToCleanReset)
	#87 FPKstartTrig:RS(SET: pin 1, RESET1: #93)
	out 1 "запуск/старт ФПК" <= #87.Q1
	#88 FPKstopTimer:TOF(IN: pin 1, PT: pin 2)
	#89 FPKstopFtrig:F_TRIG(CLK: #88.Q)
	#90 AND(#87.Q1, #91)
	#91 NOT(pin 11)
	#92 AND(#87.Q1, #94.Q, #96)
	out 2 "ФПК не стартовал" <= #92
	#93 OR(#89.Q, pin 4, pin 5, #95, #97, #100.Q1)
	#94 FPKnotStartedTimer:TON(IN: #90, PT: pin 10)
	#95 NOT(pin 3)
	#96 NOT(pin 9)
	#97 NOT(pin 6)
	#98 AND(#87.Q1, #99)
	#99 GE(pin 7, pin 8)
	#100 FPKneedToCleanTrig:RS(SET: #98, RESET1: #86.Q)
	out 3 "ФПК нужно почистить!" <= #100.Q1
	#101 S FPKneedToCleanReset <= #100.Q1
	#102 FPKneedToCleanResetRtrig:R_TRIG(CLK: pin 6)
	#103 R FPKneedToCleanReset <= #102.Q
END_MACRO
#104 DD1_DO10 <= #85.out 1
#105 FPKnotStarted <= #85.out 2
#106 FPKneedToClean <= #85.out 3
#107 MACRO контроль аналогового входа DD1_AI3(pin 1 "вход": DD1_AI3)
	(* Не смотрим конкретную ошибку, / определяем,что вход неисправен без расшифровки. *)
	#108 DD1_AI3_QE0101:DECODE_FLOAT(VALUE: pin 1, DEF_VALUE: -)
	#109 NE(#108._ERR, 0)
	out 2 "авария" <= #109
	out 1 "выход" <= #108.OUT_VALUE
END_MACRO
#110 DD1_AI3_QE0101value <= #107.out 1
#111 DD1_AI3_error <= #107.out 2
#112 MACRO контроль аналогового входа DD1_AI4(pin 1 "вход": DD1_AI4)
	(* Не смотрим конкретную ошибку, / определяем,что вход неисправен без расшифровки. *)
	#113 DD1_AI4_QE0102:DECODE_FLOAT(VALUE: pin 1, DEF_VALUE: -)
	#114 NE(#113._ERR, 0)
	out 2 "авария" <= #114
	out 1 "выход" <= #113.OUT_VALUE
END_MACRO
#115 DD1_AI4_QE0102value <= #112.out 1
#116 DD1_AI4_error <= #112.out 2
#117 MACRO контроль аналогового входа DD1_AI5(pin 1 "вход": DD1_AI5)
	(* Не смотрим конкретную ошибку, / определяем,что вход неисправен без расшифровки. *)
	#118 DD1_AI5_FPK:DECODE_FLOAT(VALUE: pin 1, DEF_VALUE: -)
	#119 NE(#118._ERR, 0)
	out 2 "авария" <= #119
	out 1 "выход" <= #118.OUT_VALUE
END_MACRO
#120 DD1_AI5_FPKpressureValue <= #117.out 1
#121 DD1_AI5_error <= #117.out 2
#122 MACRO управление НД05.02 УПГ(pin 1 "вход расходомера в куб/час": DD1_AI1_FT0101value, pin 2 "max производительность НД в мл/мин": ND0502setMaxDosVal, pin 3 "задание дозирования в мл/куб": ND0502setKoefProp, pin 4 "режим:1 насос главный": ND0502regimeP1M, pin 5 "режим: 2 насос главный": ND0502regimeP2M, pin 6 "режим: по наработке": ND0502regimeByWT, pin 7 "режим: по кол-ву включений": ND0502regimeByC, pin 8 "авария 1 насоса": DD6_DI.0, pin 9 "авария 2 насоса": DD6_DI.1, pin 10 "сброс аварий": alarmReset, pin 11 "сброс счетчика включений 1 насоса": ND0502resetCountP1, pin 12 "сброс ссчетчика включений 2 насоса": ND0502resetCountP2, pin 13 "сброс наработки 1 насоса": ND0502resetWorkTimeP1, pin 14 "сброс наработки 2 насоса": ND0502resetWorkTimeP2)
	(* сигнал 4...20мА на НД05.02/02 *)
	(* сигнал 4...20мА на НД05.02/01 *)
	(* Если на входе SEL = TRUE, / то нижнее значение, / иначе - то,что посередине. *)
	#123 SEL(#130.pump1ON, 4, #124.outputValue)
	out 6 "выход 4...20мА насоса 1" <= #123
	#124 ND0502dosing:DosingPumpProportional(flowValue: pin 1, setMinPumpDosingValue: -, setMaxPumpDosingValue: pin 2, minOutputValue: -, maxOutputValue: -, setKoeffProportionality: pin 3, minFlowToStart: -)
	out 1 "ошибка блока дозирования" <= #124.dosingError
	#125 SEL(#130.pump2ON, 4, #124.outputValue)
	#126 linTrafo050202:LIN_TRAFO(IN: #125, IN_MIN: 4, IN_MAX: 20, OUT_MIN: 0, OUT_MAX: 1000)
	#127 REAL_TO_WORD(#126.OUT)
	out 7 "выход 4...20мА насоса 2" <= #127
	#128 ND0502regime:choosePumpRegime(start: #124.startDosingPump, pump1Main: pin 4, pump2Main: pin 5, byCounter: #129, byWorkTime: pin 6)
	out 2 "статус: 1 насос главный" <= #128.pump1MainActive
	out 3 "статус: 2 насос главный" <= #128.pump2MainActive
	out 4 "статус: по кол-ву включений" <= #128.byCounterActive
	#129 OR(pin 7, startInitializer)
	out 5 "статус: по наработке" <= #128.byWorkTimeActive
	#130 ND0502manager:TwoPumpManager(startStopPump1: #128.startPump1, startStopPump2: #128.startPump2, alarmPump1: #131, alarmPump2: #132, alarmReset: pin 10, counterStart: #128.startByCounter, Pump1ResetCounter: pin 11, Pump2ResetCounter: pin 12, ValueToResetCounter: -, workTimeStart: #128.startByWorkTime, workTimePump1Reset: pin 13, workTimePump2Reset: pin 14)
	out 12 "сигнал на включение насоса 1" <= #130.pump1ON
	#131 NOT(pin 8)
	out 13 "сигнал на включение насоса 2" <= #130.pump2ON
	out 8 "счетчик включений насоса 1" <= #130.counterPump1
	#132 NOT(pin 9)
	out 9 "счетчик включений насоса 2" <= #130.counterPump2
	out 10 "счетчик наработки насоса 1" <= #130.currentWorkTimePump1
	out 11 "счетчик наработки насоса 2" <= #130.currentWorkTimePump2
END_MACRO
#133 ND0502dosingError <= #122.out 1
#134 ND0502statRegimeP1M <= #122.out 2
#135 ND0502statRegimeP2M <= #122.out 3
#136 ND0502statRegimeByC <= #122.out 4
#137 ND0502statRegimeByWT <= #122.out 5
#138 DD1_AO3 <= #122.out 6
#139 DD10_AO0 <= #122.out 7
#140 ND0502counterP1 <= #122.out 8
#141 ND0502counterP2 <= #122.out 9
#142 ND0502workTimeP1 <= #122.out 10
#143 ND0502workTimeP2 <= #122.out 11
#144 DD4_DO.4 <= #122.out 12
#145 DD4_DO.5 <= #122.out 13
#146 AND(DD2_DO.1, DD5_DI.4)
#147 N0105statStartedP1 <= #146
#148 AND(DD5_DI.4, DD2_DO.2)
#149 N0105statStartedP2 <= #148
#150 MACRO Наполнение РЧВ02.03 (заслонка ЗДЭ02.25)(pin 1 "LS02.02раб.верх.уровень РЧВ": DD6_DI.14, pin 2 "LSA02.01 Перелив РЧВ": DD6_DI.13, pin 3 "статус ЗДЭ02.25 открыт": DD9_DI.0, pin 4 "статус ЗДЭ02.25 закрыт": DD9_DI.1, pin 5 "сброс аварий": alarmReset, pin 6 "время на открытие/закрытие": timeToOpenCloseValve)
	#151 OR(testZDE0225, pin 1)
	#152 NOT(pin 1)
	#153 ZDE0225:SimpleValve(inputOpen: #151, inputClose: #154, statusOpen: pin 3, statusClose: pin 4, reset: pin 5, timeToOpenClose: pin 6)
	out 1 "выход на открытие ЗДЭ02.25" <= #153.outputOpen
	#154 OR(#152, #155)
	out 2 "выход на закрытие ЗДЭ02.25" <= #153.outputClose
	out 3 "авария на открытие ЗДЭ02.25" <= #153.errorToOpen
	#155 NOT(pin 2)
	out 4 "авария на закрытие ЗДЭ02.25" <= #153.errorToClose
END_MACRO
#156 DD4_DO.0 <= #150.out 1
#157 DD4_DO.1 <= #150.out 2
#158 ZDE0225errorToOpen <= #150.out 3
#159 ZDE0225errorToClose <= #150.out 4
#160 MACRO управление Н02.04 (подача из РЧВ)(pin 1 "промывка ФС02.01/01": DD6_DI.20, pin 2 "промывка ФС02.01/02": DD6_DI.22, pin 3 "промывка ФС02.01/03": DD6_DI.24, pin 4 "промывка ФС02.01/04": DD6_DI.26, pin 5 "промывка ФС02.01/05": DD6_DI.28, pin 6 "промывка ФС02.01/06": DD6_DI.30, pin 7 "промывка ФС02.02/01": DD7_DI.0, pin 8 "промывка ФС02.02/02": DD7_DI.2, pin 9 "промывка ФС02.02/03": DD7_DI.4, pin 10 "промывка ФС02.02/04": DD7_DI.6, pin 11 "промывка ФС02.02/05": DD7_DI.8, pin 12 "промывка ФС02.02/06": DD7_DI.10, pin 13 "открыт КЭМ05.01": DD1_DI11, pin 14 "открыт КЭМ06.01": DD1_DI10, pin 15 "открыт КЭМ07.01": DD1_DI9, pin 16 "открыт КЭМ08.01": DD1_DI8, pin 17 "сухой ход Н02.04 (0=сух.ход)": DD5_DI.11, pin 18 "выбрать режим: Н02.04/01 - главный": N0204regimeP1M, pin 19 "выбрать режим: Н02.04/02 - главный": N0204regimeP2M, pin 20 "выбрать режим: по кол-ву включений": N0204regimeByC, pin 21 "выбрать режим: по наработке": N0204regimeWT, pin 22 "авария Н02.04/01 (0=авария)": DD5_DI.7, pin 23 "авария Н02.04/02 (0=авария)": DD5_DI.8, pin 24 "сброс аварий": alarmReset, pin 25 "сброс счетчика включений Н02.04/01": N0204resetCountP1, pin 26 "сброс счетчика включений Н02.04/02": N0204resetCountP2, pin 27 "сброс счетчика наработки Н02.04/01": N0204resetWorkTimeP1, pin 28 "сброс счетчика наработки Н02.04/02": N0204resetWorkTimeP2)
	(* Проверка, что фильтры 1 / ступени в регенерации (промывке) *)
	(* Проверка, что фильтры 2 / ступени в регенерации (промывке) *)
	(* Удержание сигнала на выключение насосов для / гарантированного сброса самоподхвата реле. *)
	(* Контроль открытия хотя бы одного из клапанов КЭМ *)
	(* сброс самоподхвата реле *)
	(* Защита от сухого хода Н02.04 / (LS02.03) 0=сух.ход *)
	#161 OR(pin 1, pin 2, pin 3, pin 4, pin 5, pin 6)
	#162 OR(#161, #163, #164)
	#163 OR(pin 7, pin 8, pin 9, pin 10, pin 11, pin 12)
	#164 OR(pin 13, pin 14, pin 15, pin 16)
	#165 N020401fTrigStop:F_TRIG(CLK: #172.pump1ON)
	#166 AND(#162, pin 17)
	#167 OR(#165.Q, #170.Q)
	#168 N0204stop:TOF(IN: #167, PT: T#1s)
	out 5 "стоп Н02.04" <= #168.Q
	#169 N0204chooseRegime:choosePumpRegime(start: #166, pump1Main: pin 18, pump2Main: pin 19, byCounter: #171, byWorkTime: pin 21)
	out 1 "выбран режим Н02.04/01 = главный" <= #169.pump1MainActive
	#170 N020402fTrigStop:F_TRIG(CLK: #172.pump2ON)
	out 2 "выбран режим Н02.04/02 = главный" <= #169.pump2MainActive
	out 3 "выбран режим по кол-ву включений" <= #169.byCounterActive
	#171 OR(pin 20, startInitializer)
	out 4 "выбран режим по наработке" <= #169.byWorkTimeActive
	#172 N0204manager:TwoPumpManager(startStopPump1: #169.startPump1, startStopPump2: #169.startPump2, alarmPump1: NOT pin 22, alarmPump2: NOT pin 23, alarmReset: pin 24, counterStart: #169.startByCounter, Pump1ResetCounter: pin 25, Pump2ResetCounter: pin 26, ValueToResetCounter: -, workTimeStart: #169.startByWorkTime, workTimePump1Reset: pin 27, workTimePump2Reset: pin 28)
	out 6 "пуск Н02.04/01" <= #172.pump1ON
	out 7 "пуск Н02.04/02" <= #172.pump2ON
	out 8 "счетчик включений Н02.04/01" <= #172.counterPump1
	out 9 "счетчик включений Н02.04/02" <= #172.counterPump2
	out 10 "счетчик наработки Н02.04/01" <= #172.currentWorkTimePump1
	out 11 "счетчик наработки Н02.04/02" <= #172.currentWorkTimePump2
END_MACRO
#173 N0204statRegimeP1M <= #160.out 1
#174 N0204statRegimeP2M <= #160.out 2
#175 N0204statRegimeByC <= #160.out 3
#176 N0204statRegimeWT <= #160.out 4
#177 DD4_DO.14 <= #160.out 5
#178 DD1_DO1 <= #160.out 6
#179 DD1_DO2 <= #160.out 7
#180 N0204counterP1 <= #160.out 8
#181 N0204counterP2 <= #160.out 9
#182 N0204workTimeP1 <= #160.out 10
#183 N0204workTimeP2 <= #160.out 11
#184 MACRO управление НД06.02 УПК(pin 1 "вход расходомера в куб/час": DD1_AI2_FT0102value, pin 2 "max производительность НД в мл/мин": ND0602setMaxDosVal, pin 3 "задание дозирования в мл/куб": ND0602setKoefProp, pin 4 "режим:1 насос главный": ND0602regimeP1M, pin 5 "режим: 2 насос главный": ND0602regimeP2M, pin 6 "режим: по наработке": ND0602regimeByWT, pin 7 "режим: по кол-ву включений": ND0602regimeByC, pin 8 "авария 1 насоса": DD6_DI.2, pin 9 "авария 2 насоса": DD6_DI.3, pin 10 "сброс аварий": alarmReset, pin 11 "сброс счетчика включений 1 насоса": ND0602resetCountP1, pin 12 "сброс ссчетчика включений 2 насоса": ND0602resetCountP2, pin 13 "сброс наработки 1 насоса": ND0602resetWorkTimeP1, pin 14 "сброс наработки 2 насоса": ND0602resetWorkTimeP2)
	(* сигнал 4...20мА на НД06.02/02 *)
	(* сигнал 4...20мА на НД06.02/01 *)
	(* Если на входе SEL = TRUE, / то нижнее значение, / иначе - то,что посередине. *)
	#185 SEL(#194.pump1ON, 4, #188.outputValue)
	#186 linTraf060201:LIN_TRAFO(IN: #185, IN_MIN: 4, IN_MAX: 20, OUT_MIN: 0, OUT_MAX: 1000)
	#187 REAL_TO_WORD(#186.OUT)
	out 6 "выход 4...20мА насоса 1" <= #187
	#188 ND0602dosing:DosingPumpProportional(flowValue: pin 1, setMinPumpDosingValue: -, setMaxPumpDosingValue: pin 2, minOutputValue: -, maxOutputValue: -, setKoeffProportionality: pin 3, minFlowToStart: -)
	out 1 "ошибка блока дозирования" <= #188.dosingError
	#189 SEL(#194.pump2ON, 4, #188.outputValue)
	#190 linTraf060202:LIN_TRAFO(IN: #189, IN_MIN: 4, IN_MAX: 20, OUT_MIN: 0, OUT_MAX: 1000)
	#191 REAL_TO_WORD(#190.OUT)
	out 7 "выход 4...20мА насоса 2" <= #191
	#192 ND0602regime:choosePumpRegime(start: #188.startDosingPump, pump1Main: pin 4, pump2Main: pin 5, byCounter: #193, byWorkTime: pin 6)
	out 2 "статус: 1 насос главный" <= #192.pump1MainActive
	out 3 "статус: 2 насос главный" <= #192.pump2MainActive
	out 4 "статус: по кол-ву включений" <= #192.byCounterActive
	#193 OR(pin 7, startInitializer)
	out 5 "статус: по наработке" <= #192.byWorkTimeActive
	#194 ND0602manager:TwoPumpManager(startStopPump1: #192.startPump1, startStopPump2: #192.startPump2, alarmPump1: #195, alarmPump2: #196, alarmReset: pin 10, counterStart: #192.startByCounter, Pump1ResetCounter: pin 11, Pump2ResetCounter: pin 12, ValueToResetCounter: -, workTimeStart: #192.startByWorkTime, workTimePump1Reset: pin 13, workTimePump2Reset: pin 14)
	out 12 "сигнал на включение насоса 1" <= #194.pump1ON
	#195 NOT(pin 8)
	out 13 "сигнал на включение насоса 2" <= #194.pump2ON
	out 8 "счетчик включений насоса 1" <= #194.counterPump1
	#196 NOT(pin 9)
	out 9 "счетчик включений насоса 2" <= #194.counterPump2
	out 10 "счетчик наработки насоса 1" <= #194.currentWorkTimePump1
	out 11 "счетчик наработки насоса 2" <= #194.currentWorkTimePump2
END_MACRO
#197 ND0602dosingError <= #184.out 1
#198 ND0602statRegimeP1M <= #184.out 2
#199 ND0602statRegimeP2M <= #184.out 3
#200 ND0602statRegimeByC <= #184.out 4
#201 ND0602statRegimeByWT <= #184.out 5
#202 DD10_AO1 <= #184.out 6
#203 DD10_AO2 <= #184.out 7
#204 ND0602counterP1 <= #184.out 8
#205 ND0602counterP2 <= #184.out 9
#206 ND0602workTimeP1 <= #184.out 10
#207 ND0602workTimeP2 <= #184.out 11
#208 DD4_DO.6 <= #184.out 12
#209 DD4_DO.7 <= #184.out 13
#210 OR(errorToOpenZDE0301, errorToCloseZDE0301, errorToOpenZDE0302, errorToCloseZDE0302)
#211 OR(DD5_DI.27, #210)
#212 OR(#210, DD5_DI.29)
#213 MACRO Работа УФО03.01(pin 1 "Работа УФО03.01/01": DD5_DI.26, pin 2 "Работа УФО03.01/02": DD5_DI.28, pin 3 "Значение расхода от FT01.02": DD1_AI2_FT0102value, pin 4 "мин.допустимый расход для насосов Н01.05": N0105minFlow, pin 5 "Задержка включения УФО на создание потока": UFO0301startDelayTime, pin 6 "выбор режим: УФО03.01/01 главное": UFO0301regimeP1M, pin 7 "выбор режим: УФО03.01/02 главное": UFO0301regimeP2M, pin 8 "выбор режим: по кол-ву включений": UFO0301regimeByC, pin 9 "выбор режим: по наработке": UFO0301regimeWT, pin 10 "авария УФО03.01/01": #211, pin 11 "авария УФО03.01/02": #212, pin 12 "сброс аварий": alarmReset, pin 13 "сброс счетчика включений УФО03.01/01": UFO0301resetCountP1, pin 14 "сброс счетчика включений УФО03.01/02": UFO0301resetCountP2, pin 15 "сброс счетчика наработки УФО03.01/01": UFO0301resetWorkTimeP1, pin 16 "сброс счетчика наработки УФО03.01/02": UFO0301resetWorkTimeP2)
	(* Контроль, если УФО включили вручную, / а потока при этом нет. *)
	(* Для подачи предостережения на пульте / оператора (при необходимости), а также / сигнализации лампой АВАРИЯ. *)
	(* Задержка старта УФО *)
	(* Включаем УФО, если расходомер показывает расход больше, / чем заданный как минимально допустимый для работы насосов Н01.05. *)
	#214 OR(pin 1, pin 2)
	#215 AND(#214, #216)
	out 1 "УФО вкл без потока" <= #215
	#216 NOT(#218.Q)
	#217 GE(pin 3, pin 4)
	#218 UFO0301startDelay:TON(IN: #217, PT: pin 5)
	#219 UFO0301regimeManager:choosePumpRegime(start: #218.Q, pump1Main: pin 6, pump2Main: pin 7, byCounter: #220, byWorkTime: pin 9)
	out 2 "активен режим - главное УФО 03.01/01" <= #219.pump1MainActive
	out 3 "активен режим - главное УФО 03.01/02" <= #219.pump2MainActive
	out 4 "активен режим - по кол-ву включений" <= #219.byCounterActive
	#220 OR(startInitializer, pin 8)
	out 5 "активен режим - по наработке" <= #219.byWorkTimeActive
	#221 UFO0301manager:TwoPumpManager(startStopPump1: #219.startPump1, startStopPump2: #219.startPump2, alarmPump1: pin 10, alarmPump2: pin 11, alarmReset: pin 12, counterStart: #219.startByCounter, Pump1ResetCounter: pin 13, Pump2ResetCounter: pin 14, ValueToResetCounter: -, workTimeStart: #219.startByWorkTime, workTimePump1Reset: pin 15, workTimePump2Reset: pin 16)
	out 6 "авт. пуск УФО03.01/01" <= #221.pump1ON
	out 7 "авт. пуск УФО03.01/02" <= #221.pump2ON
	out 8 "счетчик включений УФО03.01/01" <= #221.counterPump1
	out 9 "счетчик включений УФО03.01/02" <= #221.counterPump2
	out 10 "счетчик наработки УФО03.01/01" <= #221.currentWorkTimePump1
	out 11 "счетчик наработки УФО03.01/02" <= #221.currentWorkTimePump2
END_MACRO
#222 UFO0301noFlowAttention <= #213.out 1
#223 UFO0301statRegimeP1M <= #213.out 2
#224 UFO0301statRegimeP2M <= #213.out 3
#225 UFO0301statRegimeByC <= #213.out 4
#226 UFO0301statRegimeWT <= #213.out 5
#227 UFO0301counterP1 <= #213.out 8
#228 UFO0301counterP2 <= #213.out 9
#229 UFO0301workTimeP1 <= #213.out 10
#230 UFO0301workTimeP2 <= #213.out 11
#231 MACRO работа задвижек перед УФО и автом.пуск(pin 1 "сигнал на пуск УФО03.01/01": #213.out 6, pin 2 "сигнал на пуск УФО03.01/02": #213.out 7)
	(* авт.пускУФО03.01/02 *)
	(* авт.пускУФО03.01/01 *)
	(* 1 = тест задвижек ЗДЭ / 0 = возможность автом.пуска УФО *)
	(* 1 = открыть ЗДЭ03.01 / 0 = закрыть ЗДЭ03.01 *)
	(* 1 = открыть ЗДЭ03.02 / 0 = закрыть ЗДЭ03.02 *)
	#232 NOT(testZDE03)
	#233 NOT(testZDE03)
	#234 AND(#232, #236, DD1_DI12)
	#235 DD1_DO8 <= #234
	#236 SEL(testZDE03, pin 1, manualZDE0301)
	#237 ZDE0301:SimpleValve(inputOpen: #236, inputClose: NOT #236, statusOpen: DD1_DI12, statusClose: DD1_DI13, reset: alarmReset, timeToOpenClose: timeToOpenCloseValve)
	#238 DD4_DO.16 <= #237.outputOpen
	#239 DD4_DO.17 <= #237.outputClose
	#240 errorToOpenZDE0301 <= #237.errorToOpen
	#241 errorToCloseZDE0301 <= #237.errorToClose
	#242 AND(#233, #244, DD1_DI14)
	#243 DD1_DO9 <= #242
	#244 SEL(testZDE03, pin 2, manualZDE0302)
	#245 ZDE0302:SimpleValve(inputOpen: #244, inputClose: NOT #244, statusOpen: DD1_DI14, statusClose: DD1_DI15, reset: alarmReset, timeToOpenClose: timeToOpenCloseValve)
	#246 DD4_DO.18 <= #245.outputOpen
	#247 DD4_DO.19 <= #245.outputClose
	#248 errorToOpenZDE0302 <= #245.errorToOpen
	#249 errorToCloseZDE0302 <= #245.errorToClose
END_MACRO
#250 MACRO управление НД06.03 УПК(pin 1 "вход расходомера в куб/час": DD1_AI1_FT0101value, pin 2 "max производительность НД в мл/мин": ND0603setMaxDosVal, pin 3 "задание дозирования в мл/куб": ND0603setKoefProp, pin 4 "режим:1 насос главный": ND0603regimeP1M, pin 5 "режим: 2 насос главный": ND0603regimeP2M, pin 6 "режим: по наработке": ND0603regimeByWT, pin 7 "режим: по кол-ву включений": ND0603regimeByC, pin 8 "авария 1 насоса": DD6_DI.4, pin 9 "авария 2 насоса": DD6_DI.5, pin 10 "сброс аварий": alarmReset, pin 11 "сброс счетчика включений 1 насоса": ND0603resetCountP1, pin 12 "сброс ссчетчика включений 2 насоса": ND0603resetCountP2, pin 13 "сброс наработки 1 насоса": ND0603resetWorkTimeP1, pin 14 "сброс наработки 2 насоса": ND0603resetWorkTimeP2)
	(* сигнал 4...20мА на НД06.03/02 *)
	(* сигнал 4...20мА на НД06.03/01 *)
	(* Если на входе SEL = TRUE, / то нижнее значение, / иначе - то,что посередине. *)
	#251 SEL(#260.pump1ON, 4, #254.outputValue)
	#252 linTraf060301:LIN_TRAFO(IN: #251, IN_MIN: 4, IN_MAX: 20, OUT_MIN: 0, OUT_MAX: 1000)
	#253 REAL_TO_WORD(#252.OUT)
	out 6 "выход 4...20мА насоса 1" <= #253
	#254 ND0603dosing:DosingPumpProportional(flowValue: pin 1, setMinPumpDosingValue: -, setMaxPumpDosingValue: pin 2, minOutputValue: -, maxOutputValue: -, setKoeffProportionality: pin 3, minFlowToStart: -)
	out 1 "ошибка блока дозирования" <= #254.dosingError
	#255 SEL(#260.pump2ON, 4, #254.outputValue)
	#256 linTraf060302:LIN_TRAFO(IN: #255, IN_MIN: 4, IN_MAX: 20, OUT_MIN: 0, OUT_MAX: 1000)
	#257 REAL_TO_WORD(#256.OUT)
	out 7 "выход 4...20мА насоса 2" <= #257
	#258 ND0603regime:choosePumpRegime(start: #254.startDosingPump, pump1Main: pin 4, pump2Main: pin 5, byCounter: #259, byWorkTime: pin 6)
	out 2 "статус: 1 насос главный" <= #258.pump1MainActive
	out 3 "статус: 2 насос главный" <= #258.pump2MainActive
	out 4 "статус: по кол-ву включений" <= #258.byCounterActive
	#259 OR(pin 7, startInitializer)
	out 5 "статус: по наработке" <= #258.byWorkTimeActive
	#260 ND0603manager:TwoPumpManager(startStopPump1: #258.startPump1, startStopPump2: #258.startPump2, alarmPump1: #261, alarmPump2: #262, alarmReset: pin 10, counterStart: #258.startByCounter, Pump1ResetCounter: pin 11, Pump2ResetCounter: pin 12, ValueToResetCounter: -, workTimeStart: #258.startByWorkTime, workTimePump1Reset: pin 13, workTimePump2Reset: pin 14)
	out 12 "сигнал на включение насоса 1" <= #260.pump1ON
	#261 NOT(pin 8)
	out 13 "сигнал на включение насоса 2" <= #260.pump2ON
	out 8 "счетчик включений насоса 1" <= #260.counterPump1
	#262 NOT(pin 9)
	out 9 "счетчик включений насоса 2" <= #260.counterPump2
	out 10 "счетчик наработки насоса 1" <= #260.currentWorkTimePump1
	out 11 "счетчик наработки насоса 2" <= #260.currentWorkTimePump2
END_MACRO
#263 ND0603dosingError <= #250.out 1
#264 ND0603statRegimeP1M <= #250.out 2
#265 ND0603statRegimeP2M <= #250.out 3
#266 ND0603statRegimeByC <= #250.out 4
#267 ND0603statRegimeByWT <= #250.out 5
#268 DD10_AO3 <= #250.out 6
#269 DD10_AO4 <= #250.out 7
#270 ND0603counterP1 <= #250.out 8
#271 ND0603counterP2 <= #250.out 9
#272 ND0603workTimeP1 <= #250.out 10
#273 ND0603workTimeP2 <= #250.out 11
#274 DD4_DO.8 <= #250.out 12
#275 DD4_DO.9 <= #250.out 13
#276 MACRO управление Н04.04 (дренажные)(pin 1 "защита от сухого хода Н04.04": DD5_DI.18, pin 2 "автоматич.пускН04.04": DD5_DI.19, pin 3 "режим Н04.04/01 главный": N0404regimeP1M, pin 4 "режим Н04.04/02 главный": N0404regimeP2M, pin 5 "режим по кол-ву включений": N0404regimeByC, pin 6 "режим по наработке": N0404regimeWT, pin 7 "авария Н04.04/01": DD5_DI.15, pin 8 "авария Н04.04/02": DD5_DI.14, pin 9 "сброс аварий": alarmReset, pin 10 "сброс счетчика включений Н04.04/01": N0404resetCountP1, pin 11 "сброс счетчика включений Н04.04/02": N0404resetCountP2, pin 12 "сброс счетчика наработки Н04.04/01": N0404resetWorkTimeP1, pin 13 "сброс счетчика наработки Н04.04/02": N0404resetWorkTimeP2)
	(* сбрасывает самоподхват пускового реле *)
	(* Излишняя перестраховка по сухому ходу, / на уровне реле уже все отрабатывается. *)
	(* насосы имеют электрическую блокировку / от одновременного включения *)
	(* от поплавка *)
	(* сухой ход Н04.04 / 0=защита *)
	(* 0=авария *)
	#277 NOT(pin 1)
	out 1 "стоп Н04.04" <= #277
	#278 AND(pin 1, pin 2)
	#279 N0401choosePumpRegime:choosePumpRegime(start: #278, pump1Main: pin 3, pump2Main: pin 4, byCounter: #280, byWorkTime: pin 6)
	out 2 "выбран режим: Н04.04/01 главный" <= #279.pump1MainActive
	out 3 "выбран режим: Н04.04/02 главный" <= #279.pump2MainActive
	out 4 "выбран режим: по кол-ву включений" <= #279.byCounterActive
	#280 OR(startInitializer, pin 5)
	out 5 "выбран режим: по наработке" <= #279.byWorkTimeActive
	#281 N0404twoPumpManager:TwoPumpManager(startStopPump1: #279.startPump1, startStopPump2: #279.startPump2, alarmPump1: #282, alarmPump2: #283, alarmReset: pin 9, counterStart: #279.startByCounter, Pump1ResetCounter: pin 10, Pump2ResetCounter: pin 11, ValueToResetCounter: -, workTimeStart: #279.startByWorkTime, workTimePump1Reset: pin 12, workTimePump2Reset: pin 13)
	out 6 "пуск Н04.04/01" <= #281.pump1ON
	#282 NOT(pin 7)
	out 7 "пуск Н04.04/02" <= #281.pump2ON
	out 8 "счетчик кол-ва включений Н04.04/01" <= #281.counterPump1
	#283 NOT(pin 8)
	out 9 "счетчик кол-ва включений Н04.04/02" <= #281.counterPump2
	out 10 "счетчик времени наработки Н04.04/01" <= #281.currentWorkTimePump1
	out 11 "счетчик времени наработки Н04.04/02" <= #281.currentWorkTimePump2
END_MACRO
#284 DD4_DO.15 <= #276.out 1
#285 N0404statRegimeP1M <= #276.out 2
#286 N0404statRegimeP2M <= #276.out 3
#287 N0404statRegimeByC <= #276.out 4
#288 N0404statRegimeWT <= #276.out 5
#289 DD1_DO5 <= #276.out 6
#290 DD1_DO6 <= #276.out 7
#291 N0404counterP1 <= #276.out 8
#292 N0404counterP2 <= #276.out 9
#293 N0404workTimeP1 <= #276.out 10
#294 N0404workTimeP2 <= #276.out 11
#295 MACRO управление НД07.03 УПЩ (поддержка рН, ПИД-регулятор)(pin 1 "вход рН-метра QE01.01": DD1_AI3_QE0101value, pin 2 "уставка рН": ND0703pHsetValue, pin 3 "режим:1 насос главный": ND0703regimeP1M, pin 4 "режим: 2 насос главный": ND0703regimeP2M, pin 5 "режим: по наработке": ND0703regimeByWT, pin 6 "режим: по кол-ву включений": ND0703regimeByC, pin 7 "авария 1 насоса": DD6_DI.6, pin 8 "авария 2 насоса": DD6_DI.7, pin 9 "сброс аварий": alarmReset, pin 10 "сброс счетчика включений 1 насоса": ND0703resetCountP1, pin 11 "сброс счетчика включений 2 насоса": ND0703resetCountP2, pin 12 "сброс наработки 1 насоса": ND0703resetWorkTimeP1, pin 13 "сброс наработки 2 насоса": ND0703resetWorkTimeP2, pin 14 "ручное управл.выходом Y (4...20мА)": ND0703YoutManual, pin 15 "1=ручное/0=автомат.управл.": ND0703YmanAuto, pin 16 "вход расходомера FT01.01 (куб.м/час)": DD1_AI1_FT0101value, pin 17 "коэфф.I": ND0703koeffI, pin 18 "коэфф.D": ND0703koeffD, pin 19 "коэфф.Р": ND0703koeffP)
	(* сигнал 4...20мА на НД07.03/02 *)
	(* сигнал 4...20мА на НД07.03/01 *)
	(* Если на входе SEL = TRUE, / то нижнее значение, / иначе - то,что посередине. *)
	(* min расход в кубометрах в час / для неачала дозирования. *)
	#296 ND0703pidReg:PID(ACTUAL: pin 1, SET_POINT: pin 2, KP: pin 19, TN: pin 17, TV: pin 18, Y_MANUAL: pin 14, Y_OFFSET: 500, Y_MIN: 0, Y_MAX: 1000, MANUAL: pin 15, RESET: #296.OVERFLOW)
	#297 SEL(#304.pump1ON, 0, #296.Y)
	#298 REAL_TO_WORD(#297)
	out 5 "выход 4...20мА насоса 1" <= #298
	#299 SEL(#304.pump2ON, 0, #296.Y)
	#300 REAL_TO_WORD(#299)
	out 6 "выход 4...20мА насоса 2" <= #300
	#301 GE(pin 16, 10)
	#302 ND0703regime:choosePumpRegime(start: #301, pump1Main: pin 3, pump2Main: pin 4, byCounter: #303, byWorkTime: pin 5)
	out 1 "статус: 1 насос главный" <= #302.pump1MainActive
	out 2 "статус: 2 насос главный" <= #302.pump2MainActive
	out 3 "статус: по кол-ву включений" <= #302.byCounterActive
	out 4 "статус: по наработке" <= #302.byWorkTimeActive
	#303 OR(pin 6, startInitializer)
	#304 ND0703manager:TwoPumpManager(startStopPump1: #302.startPump1, startStopPump2: #302.startPump2, alarmPump1: #305, alarmPump2: #306, alarmReset: pin 9, counterStart: #302.startByCounter, Pump1ResetCounter: pin 10, Pump2ResetCounter: pin 11, ValueToResetCounter: -, workTimeStart: #302.startByWorkTime, workTimePump1Reset: pin 12, workTimePump2Reset: pin 13)
	out 11 "сигнал на включение насоса 1" <= #304.pump1ON
	#305 NOT(pin 7)
	out 12 "сигнал на включение насоса 2" <= #304.pump2ON
	out 7 "счетчик включений насоса 1" <= #304.counterPump1
	#306 NOT(pin 8)
	out 8 "счетчик включений насоса 2" <= #304.counterPump2
	out 9 "счетчик наработки насоса 1" <= #304.currentWorkTimePump1
	out 10 "счетчик наработки насоса 2" <= #304.currentWorkTimePump2
END_MACRO
#307 ND0703statRegimeP1M <= #295.out 1
#308 ND0703statRegimeP2M <= #295.out 2
#309 ND0703statRegimeByC <= #295.out 3
#310 ND0703statRegimeByWT <= #295.out 4
#311 DD10_AO5 <= #295.out 5
#312 DD10_AO6 <= #295.out 6
#313 ND0703counterP1 <= #295.out 7
#314 ND0703counterP2 <= #295.out 8
#315 ND0703workTimeP1 <= #295.out 9
#316 ND0703workTimeP2 <= #295.out 10
#317 DD4_DO.10 <= #295.out 11
#318 DD4_DO.11 <= #295.out 12
#319 MACRO импульсный счетчик FQS0301(pin 1 "вход от счетчика": DD6_DI.19, pin 2 "вес импульса счетчика": FQS0301impulsValue, pin 3 "сброс счетчика": FQS0301reset, pin 4 "величина коррекции счетчика": FQS0301correction, pin 5 "прибавить коррекцию": FQS0301addCorrection, pin 6 "вычесть коррекцию": FQS0301deleteCorrection)
	(* сброс показаний счетчика *)
	(* значение в REAL (в какой-то момент начинает / отображаться в экспоненциальной форме) *)
	(* Если в результате коррекции накопленная сумма станет меньше нуля, то она принудительно станет равна нулю. *)
	(* коррекция показаний счетчика. *)
	(* число, коорое будем прибавлять или / вычитать из накопленной суммы стоков. *)
	#320 FQS0301rTrig:R_TRIG(CLK: pin 1)
	#321 ADD(EN: #320.Q, FQS0301totalAmount, pin 2)
	out 1 "накопленная сумма стоков (REAL)" <= #321
	#322 FQS0301resetRtrig:R_TRIG(CLK: pin 3)
	#323 MOVE(EN: #322.Q, 0)
	#324 FQS0301totalAmount <= #323
	#325 FQS0301addCorrRtrig:R_TRIG(CLK: pin 5)
	#326 ADD(EN: #325.Q, FQS0301totalAmount, pin 4)
	#327 FQS0301totalAmount <= #326
	#328 FQS0301deleteCorrRtrig:R_TRIG(CLK: pin 6)
	#329 SUB(EN: #328.Q, FQS0301totalAmount, pin 4)
	#330 FQS0301totalAmount <= #329
	#331 LT(FQS0301totalAmount, 0)
	#332 MOVE(EN: #331, 0)
	#333 FQS0301totalAmount <= #332
END_MACRO
#334 FQS0301totalAmount <= #319.out 1
#335 MACRO управление НД08.03 УПФ(pin 1 "вход расходомера в куб/час": DD1_AI1_FT0101value, pin 2 "max производительность НД в мл/мин": ND0803setMaxDosVal, pin 3 "задание дозирования в мл/куб": ND0803setKoefProp, pin 4 "режим:1 насос главный": ND0803regimeP1M, pin 5 "режим: 2 насос главный": ND0803regimeP2M, pin 6 "режим: по наработке": ND0803regimeByWT, pin 7 "режим: по кол-ву включений": ND0803regimeByC, pin 8 "авария 1 насоса": DD5_DI.12, pin 9 "авария 2 насоса": DD5_DI.13, pin 10 "сброс аварий": alarmReset, pin 11 "сброс счетчика включений 1 насоса": ND0803resetCountP1, pin 12 "сброс ссчетчика включений 2 насоса": ND0803resetCountP2, pin 13 "сброс наработки 1 насоса": ND0803resetWorkTimeP1, pin 14 "сброс наработки 2 насоса": ND0803resetWorkTimeP2, pin 15 "сухой ход 1 насоса": DD1_DI6, pin 16 "сухой ход 2 насоса": DD1_DI7)
	(* сигнал 4...20мА на НД08.03/02 *)
	(* сигнал 4...20мА на НД08.03/01 *)
	(* Если на входе SEL = TRUE, / то нижнее значение, / иначе - то,что посередине. *)
	#336 SEL(#345.pump1ON, 0, #337.outputValue)
	out 6 "выход 4...20мА насоса 1" <= #336
	#337 ND0803dosing:DosingPumpProportional(flowValue: pin 1, setMinPumpDosingValue: -, setMaxPumpDosingValue: pin 2, minOutputValue: -, maxOutputValue: -, setKoeffProportionality: pin 3, minFlowToStart: -)
	out 1 "ошибка блока дозирования" <= #337.dosingError
	#338 SEL(#345.pump2ON, 0, #337.outputValue)
	out 7 "выход 4...20мА насоса 2" <= #338
	#339 ND0803regime:choosePumpRegime(start: #337.startDosingPump, pump1Main: pin 4, pump2Main: pin 5, byCounter: #340, byWorkTime: pin 6)
	out 2 "статус: 1 насос главный" <= #339.pump1MainActive
	out 3 "статус: 2 насос главный" <= #339.pump2MainActive
	out 4 "статус: по кол-ву включений" <= #339.byCounterActive
	#340 OR(pin 7, startInitializer)
	out 5 "статус: по наработке" <= #339.byWorkTimeActive
	out 12 "сигнал на включение насоса 1" <= #345.pump1ON
	#341 NOT(pin 8)
	#342 OR(#341, pin 15)
	out 13 "сигнал на включение насоса 2" <= #345.pump2ON
	#343 NOT(pin 9)
	#344 OR(#343, pin 16)
	#345 ND0803manager:TwoPumpManager(startStopPump1: #339.startPump1, startStopPump2: #339.startPump2, alarmPump1: #342, alarmPump2: #344, alarmReset: pin 10, counterStart: #339.startByCounter, Pump1ResetCounter: pin 11, Pump2ResetCounter: pin 12, ValueToResetCounter: -, workTimeStart: #339.startByWorkTime, workTimePump1Reset: pin 13, workTimePump2Reset: pin 14)
	out 8 "счетчик включений насоса 1" <= #345.counterPump1
	out 9 "счетчик включений насоса 2" <= #345.counterPump2
	out 10 "счетчик наработки насоса 1" <= #345.currentWorkTimePump1
	out 11 "счетчик наработки насоса 2" <= #345.currentWorkTimePump2
END_MACRO
#346 ND0803dosingError <= #335.out 1
#347 ND0803statRegimeP1M <= #335.out 2
#348 ND0803statRegimeP2M <= #335.out 3
#349 ND0803statRegimeByC <= #335.out 4
#350 ND0803statRegimeByWT <= #335.out 5
#351 DD1_AO1 <= #335.out 6
#352 DD1_AO2 <= #335.out 7
#353 ND0803counterP1 <= #335.out 8
#354 ND0803counterP2 <= #335.out 9
#355 ND0803workTimeP1 <= #335.out 10
#356 ND0803workTimeP2 <= #335.out 11
#357 DD1_DO3 <= #335.out 12
#358 DD1_DO4 <= #335.out 13
#359 AND(DD1_DI5, DD1_DI4, DD6_DI.11)
#360 DD1_DO8 <= #359
#361 EQ(lastError, 0)
#362 alarmPLKnetworkDelay:TOF(IN: #361, PT: T#20s)
#363 NOT(#362.Q)
#364 alarmPLKnetwork <= #363
#365 MACRO управление НД08.04 УПФ(pin 1 "насос Н04.01 работает": DD7_DI.13, pin 2 "авария НД08.04": DD6_DI.16, pin 3 "уставкаНД08.04(0...100%)": ND0804doseValue)
	(* Преобразует сигнал 0...100 / пропорционально в 4...20мА, / в модуль АО подаем 0...1000. *)
	#366 AND(pin 1, pin 2)
	out 1 "пуск/стоп НД08.04" <= #366
	#367 ND0804linearTransformator:LIN_TRAFO(IN: pin 3, IN_MIN: 0, IN_MAX: 100, OUT_MIN: 0, OUT_MAX: 1000)
	#368 REAL_TO_WORD(#367.OUT)
	out 2 "управление НД08.04 (4...20мА)" <= #368
	out 3 "ошибка блока дозирования" <= #367.ERROR
END_MACRO
#369 DD4_DO.12 <= #365.out 1
#370 DD10_AO7 <= #365.out 2
#371 ND0804dosingError <= #365.out 3
#372 NOT(DD6_DI.0)
#373 alarmND050201 <= #372
#374 NOT(DD6_DI.23)
#375 alarmFS020102 <= #374
#376 NOT(DD9_DI.14)
#377 alarmZDE0211power <= #376
#378 NOT(DD6_DI.1)
#379 alarmND050202 <= #378
#380 NOT(DD6_DI.25)
#381 alarmFS020103 <= #380
#382 NOT(DD9_DI.15)
#383 alarmZDE0212power <= #382
#384 NOT(DD6_DI.2)
#385 alarmND060201 <= #384
#386 NOT(DD6_DI.27)
#387 alarmFS020104 <= #386
#388 NOT(DD9_DI.16)
#389 alarmZDE0213power <= #388
#390 NOT(DD6_DI.3)
#391 alarmND060202 <= #390
#392 NOT(DD6_DI.29)
#393 alarmFS020105 <= #392
#394 NOT(DD9_DI.17)
#395 alarmZDE0214power <= #394
#396 MACRO контроль включения мешалок(pin 1 "работа НД06.02/01": DD4_DO.6, pin 2 "работа НД06.02/02": DD4_DO.7, pin 3 "работа НД06.03/01": DD4_DO.8, pin 4 "работа НД06.03/02": DD4_DO.9, pin 5 "работа мешалки М06.04": DD5_DI.21, pin 6 "работа НД07.03/01": DD4_DO.10, pin 7 "работа НД07.03/02": DD4_DO.11, pin 8 "работа мешалки М07.02": DD5_DI.23, pin 9 "работа НД08.03/01": DD1_DO3, pin 10 "работа НД08.03/02": DD1_DO4, pin 11 "работа НД08.04": DD4_DO.12, pin 12 "работа мешалки М08.02": DD5_DI.25)
	#397 OR(pin 1, pin 2, pin 3, pin 4)
	#398 AND(#397, #399)
	out 1 "дозирования при выключенной М06.04" <= #398
	#399 NOT(pin 5)
	#400 OR(pin 6, pin 7)
	#401 AND(#400, #402)
	out 2 "дозирования при выключенной М07.02" <= #401
	#402 NOT(pin 8)
	#403 OR(pin 9, pin 10, pin 11)
	#404 AND(#403, #405)
	out 3 "дозирования при выключенной М08.02" <= #404
	#405 NOT(pin 12)
END_MACRO
#406 M0604attention <= #396.out 1
#407 M0702attention <= #396.out 2
#408 M0802attention <= #396.out 3
#409 NOT(DD6_DI.4)
#410 alarmND060301 <= #409
#411 NOT(DD6_DI.31)
#412 alarmFS020106 <= #411
#413 NOT(DD9_DI.18)
#414 alarmZDE0215power <= #413
#415 NOT(DD6_DI.5)
#416 alarmND060302 <= #415
#417 NOT(DD7_DI.1)
#418 alarmFS020201 <= #417
#419 NOT(DD9_DI.19)
#420 alarmZDE0216power <= #419
#421 NOT(DD6_DI.6)
#422 alarmND070301 <= #421
#423 NOT(DD7_DI.3)
#424 alarmFS020202 <= #423
#425 NOT(DD9_DI.20)
#426 alarmZDE0217power <= #425
#427 NOT(DD6_DI.7)
#428 alarmND070302 <= #427
#429 NOT(DD7_DI.5)
#430 alarmFS020203 <= #429
#431 NOT(DD9_DI.21)
#432 alarmZDE0218power <= #431
#433 NOT(DD5_DI.12)
#434 alarmND080301 <= #433
#435 NOT(DD7_DI.7)
#436 alarmFS020204 <= #435
#437 NOT(DD9_DI.22)
#438 alarmZDE0219power <= #437
#439 NOT(DD5_DI.13)
#440 alarmND080302 <= #439
#441 NOT(DD7_DI.9)
#442 alarmFS020205 <= #441
#443 NOT(DD9_DI.23)
#444 alarmZDE0220power <= #443
#445 NOT(DD6_DI.16)
#446 alarmND0804 <= #445
#447 NOT(DD7_DI.11)
#448 alarmFS020206 <= #447
#449 NOT(DD9_DI.24)
#450 alarmZDE0221power <= #449
#451 NOT(DD6_DI.11)
#452 alarmOGM0104overload <= #451
#453 NOT(DD9_DI.4)
#454 alarmZDE0201power <= #453
#455 NOT(DD9_DI.25)
#456 alarmZDE0222power <= #455
#457 MACRO переменные для обмена с панелью()
	#458 MACRO PSW регистры на передачу в панель (отображение)()
		(* PSW регистры на передачу в панель (отображение) *)
		(* panFQS0301totalAmount - переменная отображена сразу на выходе соответствующего макроса (учет очищенных стоков). / Здесь не хранится. *)
		#459 panFT0101value <= DD1_AI1_FT0101value
		#460 panQE0101value <= DD1_AI3_QE0101value
		#461 panFT0102value <= DD1_AI2_FT0102value
		#462 panQE0102value <= DD1_AI4_QE0102value
		#463 panFPKpressureValue <= DD1_AI5_FPKpressureValue
		#464 panFQS0301total <= FQS0301totalAmount
		#465 panTemperature <= temperatureValue
		#466 MACRO Время наработки и кол-во включений агрегатов()
			#467 workTimeND050201:TimeFromWorkTime(input: ND0502workTimeP1)
			#468 panND050201workDays <= #467.days
			#469 panND050201workHours <= #467.hours
			#470 panND050201workMinutes <= #467.minutes
			#471 panND050201workSeconds <= #467.seconds
			#472 workTimeND050202:TimeFromWorkTime(input: ND0502workTimeP2)
			#473 panND050202workDays <= #472.days
			#474 panND050202workHours <= #472.hours
			#475 panND050202workMinutes <= #472.minutes
			#476 panND050202workSeconds <= #472.seconds
			#477 panND0502counterP1 <= ND0502counterP1
			#478 panND0502counterP2 <= ND0502counterP2
			#479 workTimeND060201:TimeFromWorkTime(input: ND0602workTimeP1)
			#480 panND060201workDays <= #479.days
			#481 panND060201workHours <= #479.hours
			#482 panND060201workMinutes <= #479.minutes
			#483 panND060201workSeconds <= #479.seconds
			#484 workTimeND060202:TimeFromWorkTime(input: ND0602workTimeP2)
			#485 panND060202workDays <= #484.days
			#486 panND060202workHours <= #484.hours
			#487 panND060202workMinutes <= #484.minutes
			#488 panND060202workSeconds <= #484.seconds
			#489 panND0602counterP1 <= ND0602counterP1
			#490 panND0602counterP2 <= ND0602counterP2
			#491 workTimeND060301:TimeFromWorkTime(input: ND0603workTimeP1)
			#492 panND060301workDays <= #491.days
			#493 panND060301workHours <= #491.hours
			#494 panND060301workMinutes <= #491.minutes
			#495 panND060301workSeconds <= #491.seconds
			#496 workTimeND060302:TimeFromWorkTime(input: ND0603workTimeP2)
			#497 panND060302workDays <= #496.days
			#498 panND060302workHours <= #496.hours
			#499 panND060302workMinutes <= #496.minutes
			#500 panND060302workSeconds <= #496.seconds
			#501 panND0603counterP1 <= ND0603counterP1
			#502 panND0603counterP2 <= ND0603counterP2
			#503 workTimeND070301:TimeFromWorkTime(input: ND0703workTimeP1)
			#504 panND070301workDays <= #503.days
			#505 panND070301workHours <= #503.hours
			#506 panND070301workMinutes <= #503.minutes
			#507 panND070301workSeconds <= #503.seconds
			#508 workTimeND070302:TimeFromWorkTime(input: ND0703workTimeP2)
			#509 panND070302workDays <= #508.days
			#510 panND070302workHours <= #508.hours
			#511 panND070302workMinutes <= #508.minutes
			#512 panND070302workSeconds <= #508.seconds
			#513 panND0703counterP1 <= ND0703counterP1
			#514 panND0703counterP2 <= ND0703counterP2
			#515 workTimeND080301:TimeFromWorkTime(input: ND0803workTimeP1)
			#516 panND080301workDays <= #515.days
			#517 panND080301workHours <= #515.hours
			#518 panND080301workMinutes <= #515.minutes
			#519 panND080301workSeconds <= #515.seconds
			#520 workTimeND080302:TimeFromWorkTime(input: ND0803workTimeP2)
			#521 panND080302workDays <= #520.days
			#522 panND080302workHours <= #520.hours
			#523 panND080302workMinutes <= #520.minutes
			#524 panND080302workSeconds <= #520.seconds
			#525 panND0803counterP1 <= ND0803counterP1
			#526 panND0803counterP2 <= ND0803counterP2
			#527 workTimeN010501:TimeFromWorkTime(input: N0105workTimeP1)
			#528 panN010501workDays <= #527.days
			#529 panN010501workHours <= #527.hours
			#530 panN010501workMinutes <= #527.minutes
			#531 panN010501workSeconds <= #527.seconds
			#532 workTimeN010502:TimeFromWorkTime(input: N0105workTimeP2)
			#533 panN010502workDays <= #532.days
			#534 panN010502workHours <= #532.hours
			#535 panN010502workMinutes <= #532.minutes
			#536 panN010502workSeconds <= #532.seconds
			#537 panN0105counterP1 <= N0105counterP1
			#538 panN0105counterP2 <= N0105counterP2
			#539 workTimeN020401:TimeFromWorkTime(input: N0204workTimeP1)
			#540 panN020401workDays <= #539.days
			#541 panN020401workHours <= #539.hours
			#542 panN020401workMinutes <= #539.minutes
			#543 panN020401workSeconds <= #539.seconds
			#544 workTimeN020402:TimeFromWorkTime(input: N0204workTimeP2)
			#545 panN020402workDays <= #544.days
			#546 panN020402workHours <= #544.hours
			#547 panN020402workMinutes <= #544.minutes
			#548 panN020402workSeconds <= #544.seconds
			#549 panN0204counterP1 <= N0204counterP1
			#550 panN0204counterP2 <= N0204counterP2
			#551 workTimeN040401:TimeFromWorkTime(input: N0404workTimeP1)
			#552 panN040401workDays <= #551.days
			#553 panN040401workHours <= #551.hours
			#554 panN040401workMinutes <= #551.minutes
			#555 panN040401workSeconds <= #551.seconds
			#556 workTimeN040402:TimeFromWorkTime(input: N0404workTimeP2)
			#557 panN040402workDays <= #556.days
			#558 panN040402workHours <= #556.hours
			#559 panN040402workMinutes <= #556.minutes
			#560 panN040402workSeconds <= #556.seconds
			#561 panN0404counterP1 <= N0404counterP1
			#562 panN0404counterP2 <= N0404counterP2
			#563 workTimeUFO030101:TimeFromWorkTime(input: UFO0301workTimeP1)
			#564 panUFO030101workDays <= #563.days
			#565 panUFO030101workHours <= #563.hours
			#566 panUFO030101workMinutes <= #563.minutes
			#567 panUFO030101workSeconds <= #563.seconds
			#568 workTimeUFO030102:TimeFromWorkTime(input: UFO0301workTimeP2)
			#569 panUFO030102workDays <= #568.days
			#570 panUFO030102workHours <= #568.hours
			#571 panUFO030102workMinutes <= #568.minutes
			#572 panUFO030102workSeconds <= #568.seconds
			#573 panUFO0301counterP1 <= UFO0301counterP1
			#574 panUFO0301counterP2 <= UFO0301counterP2
		END_MACRO
	END_MACRO
	#575 MACRO PSB регистры на передачу в панель (отображение)()
		(* PSB регистры на передачу в панель (отображение) *)
		#576 MACRO 8 bit output module 1()
			#577 panStartND050201 <= DD4_DO.4
			#578 panStartND050202 <= DD4_DO.5
			#579 panStartND060201 <= DD4_DO.6
			#580 panStartND060202 <= DD4_DO.7
			#581 panStartND060301 <= DD4_DO.8
			#582 panStartND060302 <= DD4_DO.9
			#583 panStartM0604 <= DD5_DI.21
			#584 panStartND070301 <= DD4_DO.10
		END_MACRO
		#585 MACRO 8 bit output module 2()
			#586 panStartND070302 <= DD4_DO.11
			#587 panStartM0702 <= DD5_DI.23
			#588 panStartND080301 <= DD1_DO3
			#589 panStartND080302 <= DD1_DO4
			#590 panStartND0804 <= DD4_DO.12
			#591 panStartM0802 <= DD5_DI.25
			#592 panStartN020401 <= DD5_DI.9
			#593 panStartN020402 <= DD5_DI.10
		END_MACRO
		#594 MACRO 8 bit output module 3()
			#595 panStartN010501 <= N0105statStartedP1
			#596 panStartN010502 <= N0105statStartedP2
			#597 panCleanFS020101 <= DD6_DI.20
			#598 panCleanFS020102 <= DD6_DI.22
			#599 panCleanFS020103 <= DD6_DI.24
			#600 panCleanFS020104 <= DD6_DI.26
			#601 panCleanFS020105 <= DD6_DI.28
			#602 panCleanFS020106 <= DD6_DI.30
		END_MACRO
		#603 MACRO 8 bit output module 4()
			#604 panCleanFS020201 <= DD7_DI. 0
			#605 panCleanFS020202 <= DD7_DI. 2
			#606 panCleanFS020203 <= DD7_DI. 4
			#607 panCleanFS020204 <= DD7_DI. 6
			#608 panCleanFS020205 <= DD7_DI. 8
			#609 panCleanFS020206 <= DD7_DI. 10
			#610 panSludgeReady <= DD7_DI.15
			#611 panStartN0401 <= DD7_DI.13
		END_MACRO
		#612 MACRO 8 bit output module 5()
			#613 panKSHE0401open <= DD9_DI.2
			#614 panFPKready <= DD7_DI.12
			#615 panFPKneedToClean <= FPKneedToClean
			#616 panStartN040401 <= DD5_DI.16
			#617 panStartN040402 <= DD5_DI.17
			#618 panStartUFO030101 <= DD5_DI.26
			#619 panStartUFO030102 <= DD5_DI.28
			#620 panAlarm <= alarm
		END_MACRO
		#621 MACRO 8 bit output module 6()
			#622 panErrorTempSensor <= DD1_AI0_error
			#623 panErrorFT0101 <= DD1_AI1_error
			#624 panErrorFT0102 <= DD1_AI2_error
			#625 panErrorQE0102 <= DD1_AI3_error
			#626 panErrorQE0102 <= DD1_AI4_error
			#627 panAlarmHighTemp <= alarmHighTemperature
			#628 panAlarmLowTemp <= alarmLowTemperature
			#629 panND0502dosingError <= ND0502dosingError
		END_MACRO
		#630 MACRO 8 bit output module 7()
			#631 panND0602dosingError <= ND0602dosingError
			#632 panND0603dosingError <= ND0603dosingError
			#633 panND0803dosingError <= ND0803dosingError
			#634 panND0804dosingError <= ND0804dosingError
			#635 panND080301emptyAlarm <= DD1_DI6
			#636 panND080302emptyAlarm <= DD1_DI7
			#637 panN010501alarm <= N010501alarm
			#638 panN010502alarm <= N010502alarm
		END_MACRO
		#639 MACRO 8 bit output module 8()
			#640 panZDE0225errorToOpen <= ZDE0225errorToOpen
			#641 panZDE0225errorToClose <= ZDE0225errorToClose
			#642 panFPKalarm <= DD7_DI.14
			#643 panFPKnotStarted <= FPKnotStarted
			#644 panErrorFPKsensor <= DD1_AI5_error
			#645 panFPKkshe0401errorToOpen <= FPKkshe0401errorToOpen
			#646 panFPKkshe0401errorToClose <= FPKkshe0401errorToClose
			#647 panUFO030101alarm <= DD5_DI.27
		END_MACRO
		#648 MACRO 8 bit output module 9()
			#649 panUFO030102alarm <= DD5_DI.29
			#650 panFilterFailToRegen020101 <= filterFailToRegen020101
			#651 panErrorToOpenZD0201 <= errorToOpenZD0201
			#652 panErrorToCloseZD0201 <= errorToCloseZD0201
			#653 panErrorToOpenZD0207 <= errorToOpenZD0207
			#654 panErrorToCloseZD0207 <= errorToCloseZD0207
			#655 panFilterFailToRegen020102 <= filterFailToRegen020102
			#656 panErrorToOpenZD0202 <= errorToOpenZD0202
		END_MACRO
		#657 MACRO 8 bit output module 10()
			#658 panErrorToCloseZD0202 <= errorToCloseZD0202
			#659 panErrorToOpenZD0208 <= errorToOpenZD0208
			#660 panErrorToCloseZD0208 <= errorToCloseZD0208
			#661 panFilterFailToRegen020103 <= filterFailToRegen020103
			#662 panErrorToOpenZD0203 <= errorToOpenZD0203
			#663 panErrorToCloseZD0203 <= errorToCloseZD0203
			#664 panErrorToOpenZD0209 <= errorToOpenZD0209
			#665 panErrorToCloseZD0209 <= errorToCloseZD0209
		END_MACRO
		#666 MACRO 8 bit output module 11()
			#667 panFilterFailToRegen020104 <= filterFailToRegen020104
			#668 panErrorToOpenZD0204 <= errorToOpenZD0204
			#669 panErrorToCloseZD0204 <= errorToCloseZD0204
			#670 panErrorToOpenZD0210 <= errorToOpenZD0210
			#671 panErrorToCloseZD0210 <= errorToCloseZD0210
			#672 panFilterFailToRegen020105 <= filterFailToRegen020105
			#673 panErrorToOpenZD0205 <= errorToOpenZD0205
			#674 panErrorToCloseZD0205 <= errorToCloseZD0205
		END_MACRO
		#675 MACRO 8 bit output module 12()
			#676 panErrorToOpenZD0211 <= errorToOpenZD0211
			#677 panErrorToCloseZD0211 <= errorToCloseZD0211
			#678 panFilterFailToRegen020106 <= filterFailToRegen020106
			#679 panErrorToOpenZD0206 <= errorToOpenZD0206
			#680 panErrorToCloseZD0206 <= errorToCloseZD0206
			#681 panErrorToOpenZD0212 <= errorToOpenZD0212
			#682 panErrorToCloseZD0212 <= errorToCloseZD0212
			#683 panFilterFailToRegen020201 <= filterFailToRegen020201
		END_MACRO
		#684 MACRO 8 bit output module 13()
			#685 panErrorToOpenZD0213 <= errorToOpenZD0213
			#686 panErrorToCloseZD0213 <= errorToCloseZD0213
			#687 panErrorToOpenZD0219 <= errorToOpenZD0219
			#688 panErrorToCloseZD0219 <= errorToCloseZD0219
			#689 panFilterFailToRegen020202 <= filterFailToRegen020202
			#690 panErrorToOpenZD0214 <= errorToOpenZD0214
			#691 panErrorToCloseZD0214 <= errorToCloseZD0214
			#692 panErrorToOpenZD0220 <= errorToOpenZD0220
		END_MACRO
		#693 MACRO 8 bit output module 14()
			#694 panErrorToCloseZD0220 <= errorToCloseZD0220
			#695 panFilterFailToRegen020203 <= filterFailToRegen020203
			#696 panErrorToOpenZD0215 <= errorToOpenZD0215
			#697 panErrorToCloseZD0215 <= errorToCloseZD0215
			#698 panErrorToOpenZD0221 <= errorToOpenZD0221
			#699 panErrorToCloseZD0221 <= errorToCloseZD0221
			#700 panFilterFailToRegen020204 <= filterFailToRegen020204
			#701 panErrorToOpenZD0216 <= errorToOpenZD0216
		END_MACRO
		#702 MACRO 8 bit output module 15()
			#703 panErrorToCloseZD0216 <= errorToCloseZD0216
			#704 panErrorToOpenZD0222 <= errorToOpenZD0222
			#705 panErrorToCloseZD0222 <= errorToCloseZD0222
			#706 panFilterFailToRegen020205 <= filterFailToRegen020205
			#707 panErrorToOpenZD0217 <= errorToOpenZD0217
			#708 panErrorToCloseZD0217 <= errorToCloseZD0217
			#709 panErrorToOpenZD0223 <= errorToOpenZD0223
			#710 panErrorToCloseZD0223 <= errorToCloseZD0223
		END_MACRO
		#711 MACRO 8 bit output module 16()
			#712 panFilterFailToRegen020206 <= filterFailToRegen020206
			#713 panErrorToOpenZD0218 <= errorToOpenZD0218
			#714 panErrorToCloseZD0218 <= errorToCloseZD0218
			#715 panErrorToOpenZD0224 <= errorToOpenZD0224
			#716 panErrorToCloseZD0224 <= errorToCloseZD0224
			#717 panAlarmPLKnetwork <= alarmPLKnetwork
			#718 panAlarmND050201 <= alarmND050201
			#719 panAlarmND050202 <= alarmND050202
		END_MACRO
		#720 MACRO 8 bit output module 17()
			#721 panAlarmND060201 <= alarmND060201
			#722 panAlarmND060202 <= alarmND060202
			#723 panAlarmND060301 <= alarmND060301
			#724 panAlarmND060302 <= alarmND060302
			#725 panAlarmND070301 <= alarmND070301
			#726 panAlarmND070302 <= alarmND070302
			#727 panAlarmND080301 <= alarmND080301
			#728 panAlarmND080302 <= alarmND080302
		END_MACRO
		#729 MACRO 8 bit output module 18()
			#730 panAlarmND0804 <= alarmND0804
			#731 panAlarmOGM0104overload <= alarmOGM0104overload
			#732 panAlarmRCHV0203overload <= alarmRCHV0203overload
			#733 panAlarmN040402 <= alarmN040402
			#734 panAlarmN040401 <= alarmN040401
			#735 panAlarmM0604 <= alarmM0604
			#736 panAlarmM0702 <= alarmM0702
			#737 panAlarmM0802 <= alarmM0802
		END_MACRO
		#738 MACRO 8 bit output module 19()
			#739 panAlarmN020401 <= alarmN020401
			#740 panAlarmN020402 <= alarmN020402
			#741 panAlarmFS020101 <= alarmFS020101
			#742 panAlarmFS020102 <= alarmFS020102
			#743 panAlarmFS020103 <= alarmFS020103
			#744 panAlarmFS020104 <= alarmFS020104
			#745 panAlarmFS020105 <= alarmFS020105
			#746 panAlarmFS020106 <= alarmFS020106
		END_MACRO
		#747 MACRO 8 bit output module 20()
			#748 panAlarmFS020201 <= alarmFS020201
			#749 panAlarmFS020202 <= alarmFS020202
			#750 panAlarmFS020203 <= alarmFS020203
			#751 panAlarmFS020204 <= alarmFS020204
			#752 panAlarmFS020205 <= alarmFS020205
			#753 panAlarmFS020206 <= alarmFS020206
			#754 panAlarmZDE0201power <= alarmZDE0201power
			#755 panAlarmZDE0202power <= alarmZDE0202power
		END_MACRO
		#756 MACRO 8 bit output module 21()
			#757 panAlarmZDE0203power <= alarmZDE0203power
			#758 panAlarmZDE0204power <= alarmZDE0204power
			#759 panAlarmZDE0205power <= alarmZDE0205power
			#760 panAlarmZDE0206power <= alarmZDE0206power
			#761 panAlarmZDE0207power <= alarmZDE0207power
			#762 panAlarmZDE0208power <= alarmZDE0208power
			#763 panAlarmZDE0209power <= alarmZDE0209power
			#764 panAlarmZDE0210power <= alarmZDE0210power
		END_MACRO
		#765 MACRO 8 bit output module 22()
			#766 panAlarmZDE0211power <= alarmZDE0211power
			#767 panAlarmZDE0212power <= alarmZDE0212power
			#768 panAlarmZDE0213power <= alarmZDE0213power
			#769 panAlarmZDE0214power <= alarmZDE0214power
			#770 panAlarmZDE0215power <= alarmZDE0215power
			#771 panAlarmZDE0216power <= alarmZDE0216power
			#772 panAlarmZDE0217power <= alarmZDE0217power
			#773 panAlarmZDE0218power <= alarmZDE0218power
		END_MACRO
		#774 MACRO 8 bit output module 23()
			#775 panAlarmZDE0219power <= alarmZDE0219power
			#776 panAlarmZDE0220power <= alarmZDE0220power
			#777 panAlarmZDE0221power <= alarmZDE0221power
			#778 panAlarmZDE0222power <= alarmZDE0222power
			#779 panAlarmZDE0223power <= alarmZDE0223power
			#780 panAlarmZDE0224power <= alarmZDE0224power
			#781 panAlarmZDE0225power <= alarmZDE0225power
			#782 panAlarmKSHE0401power <= alarmKSHE0401power
		END_MACRO
		#783 MACRO 8 bit output module 24()
			#784 panAlarmKNS <= alarmKNS
			#785 panAlarmPowerSocketFS <= alarmPowerSocketFS
			#786 panAlarmKEMvalvesPower <= alarmKEMvalvesPower
			#787 panAlarmEmergencyPressed <= alarmEmergencyPressed
			#788 panAlarmRKF <= alarmRKF
			#789 panUFO0301noFlowAttention <= UFO0301noFlowAttention
			#790 panM0604attention <= M0604attention
			#791 panM0702attention <= M0702attention
		END_MACRO
		#792 MACRO 8 bit output module 25()
			#793 panM0802attention <= M0802attention
			#794 panStatusKNS <= DD6_DI.8
			#795 panND0502statRegimeP1M <= ND0502statRegimeP1M
			#796 panND0502statRegimeP2M <= ND0502statRegimeP2M
			#797 panND0502statRegimeByC <= ND0502statRegimeByC
			#798 panND0502statRegimeByWT <= ND0502statRegimeByWT
			#799 panND0602statRegimeP1M <= ND0602statRegimeP1M
			#800 panND0602statRegimeP2M <= ND0602statRegimeP2M
		END_MACRO
		#801 MACRO 8 bit output module 26()
			#802 panND0602statRegimeByC <= ND0602statRegimeByC
			#803 panND0602statRegimeByWT <= ND0602statRegimeByWT
			#804 panND0603statRegimeP1M <= ND0603statRegimeP1M
			#805 panND0603statRegimeP2M <= ND0603statRegimeP2M
			#806 panND0603statRegimeByC <= ND0603statRegimeByC
			#807 panND0603statRegimeByWT <= ND0603statRegimeByWT
			#808 panND0703statRegimeP1M <= ND0703statRegimeP1M
			#809 panND0703statRegimeP2M <= ND0703statRegimeP2M
		END_MACRO
		#810 MACRO 8 bit output module 27()
			#811 panND0703statRegimeByC <= ND0703statRegimeByC
			#812 panND0703statRegimeByWT <= ND0703statRegimeByWT
			#813 panND0803statRegimeP1M <= ND0803statRegimeP1M
			#814 panND0803statRegimeP2M <= ND0803statRegimeP2M
			#815 panND0803statRegimeByC <= ND0803statRegimeByC
			#816 panND0803statRegimeByWT <= ND0803statRegimeByWT
			#817 panN0105statRegimeP1M <= N0105statRegimeP1M
			#818 panN0105statRegimeP2M <= N0105statRegimeP2M
		END_MACRO
		#819 MACRO 8 bit output module 28()
			#820 panN0105statRegimeByC <= N0105statRegimeByC
			#821 panN0105statRegimeByWT <= N0105statRegimeByWT
			#822 panN0204statRegimeP1M <= N0204statRegimeP1M
			#823 panN0204statRegimeP2M <= N0204statRegimeP2M
			#824 panN0204statRegimeByC <= N0204statRegimeByC
			#825 panN0204statRegimeWT <= N0204statRegimeWT
			#826 panN0404statRegimeP1M <= N0404statRegimeP1M
			#827 panN0404statRegimeP2M <= N0404statRegimeP2M
		END_MACRO
		#828 MACRO 8 bit output module 29()
			#829 panN0404statRegimeByC <= N0404statRegimeByC
			#830 panN0404statRegimeWT <= N0404statRegimeWT
			#831 panUFO0301statRegimeP1M <= UFO0301statRegimeP1M
			#832 panUFO0301statRegimeP2M <= UFO0301statRegimeP2M
			#833 panUFO0301statRegimeByC <= UFO0301statRegimeByC
			#834 panUFO0301statRegimeWT <= UFO0301statRegimeWT
			#835 panZDE0225open <= DD9_DI.0
			#836 panZDE0201open <= DD7_DI.16
		END_MACRO
		#837 MACRO 8 bit output module 30()
			#838 panZDE0201close <= DD7_DI.17
			#839 panZDE0202open <= DD7_DI.18
			#840 panZDE0202close <= DD7_DI.19
			#841 panZDE0203open <= DD7_DI.20
			#842 panZDE0203close <= DD7_DI.21
			#843 panZDE0204open <= DD7_DI.22
			#844 panZDE0204close <= DD7_DI.23
			#845 panZDE0205open <= DD7_DI.24
		END_MACRO
		#846 MACRO 8 bit output module 31()
			#847 panZDE0205close <= DD7_DI.25
			#848 panZDE0206open <= DD7_DI.26
			#849 panZDE0206close <= DD7_DI.27
			#850 panZDE0207open <= DD7_DI.28
			#851 panZDE0207close <= DD7_DI.29
			#852 panZDE0208open <= DD7_DI.30
			#853 panZDE0208close <= DD7_DI.31
			#854 panZDE0209open <= DD8_DI.0
		END_MACRO
		#855 MACRO 8 bit output module 32()
			#856 panZDE0209close <= DD8_DI.1
			#857 panZDE0210open <= DD8_DI.2
			#858 panZDE0210close <= DD8_DI.3
			#859 panZDE0211open <= DD8_DI.4
			#860 panZDE0211close <= DD8_DI.5
			#861 panZDE0212open <= DD8_DI.6
			#862 panZDE0212close <= DD8_DI.7
			#863 panZDE0213open <= DD8_DI.8
		END_MACRO
		#864 MACRO 8 bit output module 33()
			#865 panZDE0213close <= DD8_DI.9
			#866 panZDE0214open <= DD8_DI.10
			#867 panZDE0214close <= DD8_DI.11
			#868 panZDE0215open <= DD8_DI.12
			#869 panZDE0215close <= DD8_DI.13
			#870 panZDE0216open <= DD8_DI.14
			#871 panZDE0216close <= DD8_DI.15
			#872 panZDE0217open <= DD8_DI.16
		END_MACRO
		#873 MACRO 8 bit output module 34()
			#874 panZDE0217close <= DD8_DI.17
			#875 panZDE0218open <= DD8_DI.18
			#876 panZDE0218close <= DD8_DI.19
			#877 panZDE0219open <= DD8_DI.20
			#878 panZDE0219close <= DD8_DI.21
			#879 panZDE0220open <= DD8_DI.22
			#880 panZDE0220close <= DD8_DI.23
			#881 panZDE0221open <= DD8_DI.24
		END_MACRO
		#882 MACRO 8 bit output module 35()
			#883 panZDE0221close <= DD8_DI.25
			#884 panZDE0222open <= DD8_DI.26
			#885 panZDE0222close <= DD8_DI.27
			#886 panZDE0223open <= DD8_DI.28
			#887 panZDE0223close <= DD8_DI.29
			#888 panZDE0224open <= DD8_DI.30
			#889 panZDE0224close <= DD8_DI.31
			#890 panZDE0225close <= DD9_DI.1
		END_MACRO
		#891 MACRO 8 bit output module 36x()
			#892 panKSHE0401close <= DD9_DI.3
			#893 panZDE0301open <= DD1_DI12
			#894 panZDE0301close <= DD1_DI13
			#895 panZDE0302open <= DD1_DI14
			#896 panZDE0302close <= DD1_DI15
			#897 panErrorToOpenZDE0301 <= errorToOpenZDE0301
			#898 panErrorToCloseZDE0301 <= errorToCloseZDE0301
			#899 panErrorToOpenZDE0302 <= errorToOpenZDE0302
		END_MACRO
		#900 panErrorToCloseZDE0302 <= errorToCloseZDE0302
		#901 panAlarmZDE0301power <= alarmZDE0301power
		#902 panAlarmZDE0302power <= alarmZDE0302power
	END_MACRO
	#903 MACRO PFW регистры на чтение из панели (управление ПЛК)()
		#904 MUL(panTimeToOpenCloseValve, 1000)
		#905 REAL_TO_TIME(#904)
		#906 TimeToOpenCloseValve <= #905
		#907 maxTemperature <= panMaxTemperature
		#908 minTemperature <= panMinTemperature
		#909 ND0502setMaxDosVal <= panND0502setMaxDosVal
		#910 ND0502setKoefProp <= panND0502setKoefProp
		#911 ND0602setMaxDosVal <= panND0602setMaxDosVal
		#912 ND0602setKoefProp <= panND0602setKoefProp
		#913 ND0603setMaxDosVal <= panND0603setMaxDosVal
		#914 ND0603setKoefProp <= panND0603setKoefProp
		#915 ND0703pHsetValue <= panND0703pHsetValue
		#916 ND0703YoutManual <= panND0703YoutManual
		#917 ND0703koeffI <= panND0703koeffI
		#918 ND0703koeffD <= panND0703koeffD
		#919 ND0703koeffP <= panND0703koeffP
		#920 ND0803setMaxDosVal <= panND0803setMaxDosVal
		#921 ND0803setKoefProp <= panND0803setKoefProp
		#922 ND0804doseValue <= panND0804doseValue
		#923 N0105flowSetValue <= panN0105flowSetValue
		#924 N0105YoutManual <= panN0105YoutManual
		#925 N0105koeffI <= panN0105koeffI
		#926 N0105koeffD <= panN0105koeffD
		#927 N0105koeffP <= panN0105koeffP
		#928 FQS0301impulsValue <= panFQS0301impulsValue
		#929 FQS0301correction <= panFQS0301correction
		#930 MUL(panFPKtimeToWork, 1000)
		#931 REAL_TO_TIME(#930)
		#932 FPKtimeToWork <= #931
		#933 MUL(panFPKnotStartedTime, 1000)
		#934 REAL_TO_TIME(#933)
		#935 FPKnotStartedTime <= #934
		#936 FPKmaxPressureValue <= panFPKmaxPressureValue
		#937 filterValueToRegen <= panFilterValueToRegen
	END_MACRO
	#938 MACRO PSB регистры на чтение из панели (управление ПЛК)()
		(* PSB регистры на чтение из панели (управление ПЛК) *)
		#939 MACRO 8 bit input module 1()
			#1267 alarmReset <= panAlarmResetButton
			#1268 ND0502resetCountP1 <= panND0502resetCountP1
			#1269 ND0502resetCountP2 <= panND0502resetCountP2
			#1270 ND0502resetWorkTimeP1 <= panND0502resetWorkTimeP1
			#1271 ND0502resetWorkTimeP2 <= panND0502resetWorkTimeP2
			#1272 ND0502regimeP1M <= panND0502regimeP1M
			#1273 ND0502regimeP2M <= panND0502regimeP2M
			#1274 ND0502regimeByC <= panND0502regimeByC
		END_MACRO
		#940 MACRO 8 bit input module 2()
			#1275 ND0502regimeByWT <= panND0502regimeByWT
			#1276 ND0602resetCountP1 <= panND0602resetCountP1
			#1277 ND0602resetCountP2 <= panND0602resetCountP2
			#1278 ND0602resetWorkTimeP1 <= panND0602resetWorkTimeP1
			#1279 ND0602resetWorkTimeP2 <= panND0602resetWorkTimeP2
			#1280 ND0602regimeP1M <= panND0602regimeP1M
			#1281 ND0602regimeP2M <= panND0602regimeP2M
			#1282 ND0602regimeByC <= panND0602regimeByC
		END_MACRO
		#941 MACRO 8 bit input module 3()
			#1283 ND0602regimeByWT <= panND0602regimeByWT
			#1284 ND0603resetCountP1 <= panND0603resetCountP1
			#1285 ND0603resetCountP2 <= panND0603resetCountP2
			#1286 ND0603resetWorkTimeP1 <= panND0603resetWorkTimeP1
			#1287 ND0603resetWorkTimeP2 <= panND0603resetWorkTimeP2
			#1288 ND0603regimeP1M <= panND0603regimeP1M
			#1289 ND0603regimeP2M <= panND0603regimeP2M
			#1290 ND0603regimeByC <= panND0603regimeByC
		END_MACRO
		#942 MACRO 8 bit input module 4()
			#1291 ND0603regimeByWT <= panND0603regimeByWT
			#1292 ND0703resetCountP1 <= panND0703resetCountP1
			#1293 ND0703resetCountP2 <= panND0703resetCountP2
			#1294 ND0703resetWorkTimeP1 <= panND0703resetWorkTimeP1
			#1295 ND0703resetWorkTimeP2 <= panND0703resetWorkTimeP2
			#1296 ND0703regimeP1M <= panND0703regimeP1M
			#1297 ND0703regimeP2M <= panND0703regimeP2M
			#1298 ND0703regimeByC <= panND0703regimeByC
		END_MACRO
		#943 MACRO 8 bit input module 5()
			#1299 ND0703regimeByWT <= panND0703regimeByWT
			#1300 ND0703YmanAuto <= panND0703YmanAuto
			#1301 ND0803resetCountP1 <= panND0803resetCountP1
			#1302 ND0803resetCountP2 <= panND0803resetCountP2
			#1303 ND0803resetWorkTimeP1 <= panND0803resetWorkTimeP1
			#1304 ND0803resetWorkTimeP2 <= panND0803resetWorkTimeP2
			#1305 ND0803regimeP1M <= panND0803regimeP1M
			#1306 ND0803regimeP2M <= panND0803regimeP2M
		END_MACRO
		#944 MACRO 8 bit input module 6()
			#1307 ND0803regimeByC <= panND0803regimeByC
			#1308 ND0803regimeByWT <= panND0803regimeByWT
			#1309 N0105resetCountP1 <= panN0105resetCountP1
			#1310 N0105resetCountP2 <= panN0105resetCountP2
			#1311 N0105resetWorkTimeP1 <= panN0105resetWorkTimeP1
			#1312 N0105resetWorkTimeP2 <= panN0105resetWorkTimeP2
			#1313 N0105regimeByC <= panN0105regimeByC
			#1314 N0105regimeByWT <= panN0105regimeByWT
		END_MACRO
		#945 MACRO 8 bit input module 7()
			#1315 N0105YmanAuto <= panN0105YmanAuto
			#1316 N0204resetCountP1 <= panN0204resetCountP1
			#1317 N0204resetCountP2 <= panN0204resetCountP2
			#1318 N0204resetWorkTimeP1 <= panN0204resetWorkTimeP1
			#1319 N0204resetWorkTimeP2 <= panN0204resetWorkTimeP2
			#1320 N0204regimeP1M <= panN0204regimeP1M
			#1321 N0204regimeP2M <= panN0204regimeP2M
			#1322 N0204regimeByC <= panN0204regimeByC
		END_MACRO
		#946 MACRO 8 bit input module 8()
			#1323 N0204regimeWT <= panN0204regimeWT
			#1324 UFO0301resetCountP1 <= panUFO0301resetCountP1
			#1325 UFO0301resetCountP2 <= panUFO0301resetCountP2
			#1326 UFO0301resetWorkTimeP1 <= panUFO0301resetWorkTimeP1
			#1327 UFO0301resetWorkTimeP2 <= panUFO0301resetWorkTimeP2
			#1328 UFO0301regimeP1M <= panUFO0301regimeP1M
			#1329 UFO0301regimeP2M <= panUFO0301regimeP2M
			#1330 UFO0301regimeByC <= panUFO0301regimeByC
		END_MACRO
		#947 MACRO 8 bit input module 9()
			#1331 UFO0301regimeWT <= panUFO0301regimeWT
			#1332 N0404resetCountP1 <= panN0404resetCountP1
			#1333 N0404resetCountP2 <= panN0404resetCountP2
			#1334 N0404resetWorkTimeP1 <= panN0404resetWorkTimeP1
			#1335 N0404resetWorkTimeP2 <= panN0404resetWorkTimeP2
			#1336 N0404regimeP1M <= panN0404regimeP1M
			#1337 N0404regimeP2M <= panN0404regimeP2M
			#1338 N0404regimeByC <= panN0404regimeByC
		END_MACRO
		#948 MACRO 8 bit input module 10-11()
			(* одули 10 и 11 заполнены переменными для тестирования задвижек. / Здесь они не показаны, т.к. спешка. / Они вставлены напрямую в макросы управления промывкой фильтров. / testValvesFS020101 - testValvesFS020206 (PSB612-623) *)
			#1339 N0404regimeWT <= panN0404regimeWT
			#1340 FQS0301reset <= panFQS0301reset
			#1341 FQS0301addCorrection <= panFQS0301addCorrection
			#1342 FQS0301deleteCorrection <= panFQS0301deleteCorrection
		END_MACRO
		#949 testKSHE0401 <= panTestKSHE0401
		#950 testZDE0225 <= panTestZDE0225
		#951 testZDE03 <= panTestZDE03
		#952 manualZDE0301 <= panManualZDE0301
		#953 manualZDE0302 <= panManualZDE0302
	END_MACRO
END_MACRO
#954 NOT(DD6_DI.13)
#955 alarmRCHV0203overload <= #954
#956 NOT(DD9_DI.5)
#957 alarmZDE0202power <= #956
#958 NOT(DD9_DI.26)
#959 alarmZDE0223power <= #958
#960 MACRO переменные на диспетчеризацию()
	#961 remFT0101value <= DD1_AI1_FT0101value
	#962 remFQS0301totalAmount <= FQS0301totalAmount
	#963 remTemperatureValue <= temperatureValue
	#964 remStatusN010501started <= N0105statStartedP1
	#965 remStatusN010502started <= N0105statStartedP2
	#966 remStatusUFO030101started <= DD5_DI.26
	#967 remStatusUFO030102started <= DD5_DI.28
	#968 remAlarm <= Alarm
	#969 remN010501alarm <= N010501alarm
	#970 remN010502alarm <= N010502alarm
	#971 remFPKalarm <= DD7_DI.14
	#972 remUFO030101alarm <= DD5_DI.27
	#973 remUFO030102alarm <= DD5_DI.29
	#974 remAlarmEmergencyPressed <= alarmEmergencyPressed
	#975 remAlarmOOGM0104overload <= DD6_DI.11
	#976 remAlarmRCHV0203overload <= DD6_DI.13
END_MACRO
#977 NOT(DD5_DI.14)
#978 alarmN040402 <= #977
#979 NOT(DD9_DI.6)
#980 alarmZDE0203power <= #979
#981 NOT(DD9_DI.27)
#982 alarmZDE0224power <= #981
#983 NOT(DD5_DI.15)
#984 alarmN040401 <= #983
#985 NOT(DD9_DI.7)
#986 alarmZDE0204power <= #985
#987 NOT(DD9_DI.28)
#988 alarmZDE0225power <= #987
#989 NOT(DD5_DI.20)
#990 alarmM0604 <= #989
#991 NOT(DD9_DI.8)
#992 alarmZDE0205power <= #991
#993 NOT(DD9_DI.29)
#994 alarmKSHE0401power <= #993
#995 NOT(DD5_DI.22)
#996 alarmM0702 <= #995
#997 NOT(DD9_DI.9)
#998 alarmZDE0206power <= #997
#999 NOT(DD6_DI.9)
#1000 alarmKNS <= #999
#1001 NOT(DD5_DI.24)
#1002 alarmM0802 <= #1001
#1003 NOT(DD9_DI.10)
#1004 alarmZDE0207power <= #1003
#1005 NOT(DD6_DI.17)
#1006 alarmPowerSocketFS <= #1005
#1007 NOT(DD5_DI.7)
#1008 alarmN020401 <= #1007
#1009 NOT(DD9_DI.11)
#1010 alarmZDE0208power <= #1009
#1011 NOT(DD6_DI.18)
#1012 alarmKEMvalvesPower <= #1011
#1013 NOT(DD5_DI.8)
#1014 alarmN020402 <= #1013
#1015 NOT(DD9_DI.12)
#1016 alarmZDE0209power <= #1015
#1017 NOT(DD1_DI4)
#1018 alarmEmergencyPressed <= #1017
#1019 GT(DD1_AI2_FT0102value, 0)
#1020 filterPulserGen:PulsePerSec(start: #1019)
#1021 DIV(DD1_AI2_FT0102value, 3600)
#1022 ADD(EN: #1020.out, #1021, filterTotalAmountFT0102)
#1023 filterTotalAmountFT0102 <= #1022
#1024 NOT(DD6_DI.21)
#1025 alarmFS020101 <= #1024
#1026 NOT(DD9_DI.13)
#1027 alarmZDE0210power <= #1026
#1028 NOT(DD1_DI5)
#1029 alarmRKF <= #1028
#1030 NOT(DD9_DI.30)
#1031 alarmZDE0301power <= #1030
#1032 NOT(DD9_DI.31)
#1033 alarmZDE0302power <= #1032
#1034 MOVE(EN: filterTotalAmountReset, 0)
#1035 filterTotalAmountFT0102 <= #1034
#1036 GE(filterTotalAmountFT0102, filterValueToRegen)
#1037 MACRO управление промывкой фильтра ФС02.01.01(pin 1 "сигнал на промывку": #1036, pin 2 "авария фильтра": DD6_DI.21, pin 3 "подтверждение промывки": DD6_DI.20, pin 4 "сброс аварий": alarmReset, pin 5 "начать очередь снова": filterStartNewQueue, pin 6 "ЗДЭ02.01 открыта": DD7_DI.16, pin 7 "ЗДЭ02.01 закрыта": DD7_DI.17, pin 8 "ЗДЭ02.07 открыта": DD7_DI.28, pin 9 "ЗДЭ02.07 закрыта": DD7_DI.29, pin 10 "время движения ЗДЭ": timeToOpenCloseValve, pin 11 "авария питания ЗДЭ02.01": DD9_DI.4, pin 12 "авария питания ЗДЭ02.07": DD9_DI.10)
	(* <- выход использовать в / последнем фильтре для / начала очереди заново *)
	(* если открыт = промывка *)
	(* если открыт = фильтрация *)
	out 1 "следующий в очереди" <= #1040.output
	out 2 "промыть ФС02.01.01" <= #1039
	#1038 ZD0201:SimpleValve(inputOpen: NOT #1039, inputClose: #1039, statusOpen: pin 6, statusClose: pin 7, reset: pin 4, timeToOpenClose: pin 10)
	out 6 "открыть ЗДЭ02.01" <= #1038.outputOpen
	out 7 "закрыть ЗДЭ02.01" <= #1038.outputClose
	out 8 "авария открытия ЗДЭ02.01" <= #1038.errorToOpen
	#1039 OR(panTestValvesFS020101, #1040.regenFilterOUT)
	out 9 "авария закрытия ЗДЭ02.01" <= #1038.errorToClose
	#1040 FS020101manager:FilterQueueManager(input: pin 1, filterAlarm: #1041, regenFilterStatus: pin 3, alarmReset: pin 4, startNextLoop: pin 5)
	#1041 OR(alarmZD020107, pin 2, pin 11, pin 12)
	out 3 "ФС02.01.01 промыт" <= #1040.regenerated
	out 4 "не удалось промыть" <= #1040.failToRegen
	#1042 OR(#1038.errorToOpen, #1038.errorToClose, #1044.errorToOpen, #1044.errorToClose)
	#1043 alarmZD020107 <= #1042
	out 5 "сброс счетчика" <= #1040.counterReset
	#1044 ZD0207:SimpleValve(inputOpen: #1039, inputClose: NOT #1039, statusOpen: pin 8, statusClose: pin 9, reset: pin 4, timeToOpenClose: pin 10)
	out 10 "открыть ЗДЭ02.07" <= #1044.outputOpen
	out 11 "закрыть ЗДЭ02.07" <= #1044.outputClose
	out 12 "авария открытия ЗДЭ02.07" <= #1044.errorToOpen
	out 13 "авария закрытия ЗДЭ02.07" <= #1044.errorToClose
END_MACRO
#1045 DD2_DO.4 <= #1037.out 2
#1046 regeneratedFS020101 <= #1037.out 3
#1047 filterFailToRegen020101 <= #1037.out 4
#1048 filterTotalAmountReset <= #1037.out 5
#1049 DD2_DO.16 <= #1037.out 6
#1050 DD2_DO.17 <= #1037.out 7
#1051 errorToOpenZD0201 <= #1037.out 8
#1052 errorToCloseZD0201 <= #1037.out 9
#1053 DD2_DO.28 <= #1037.out 10
#1054 DD2_DO.29 <= #1037.out 11
#1055 errorToOpenZD0207 <= #1037.out 12
#1056 errorToCloseZD0207 <= #1037.out 13
#1057 MACRO управление промывкой фильтра ФС02.01.02(pin 1 "сигнал на промывку": #1037.out 1, pin 2 "авария фильтра": DD6_DI.23, pin 3 "подтверждение промывки": DD6_DI.22, pin 4 "сброс аварий": alarmReset, pin 5 "начать очередь снова": filterStartNewQueue, pin 6 "ЗДЭ02.02 открыта": DD7_DI.18, pin 7 "ЗДЭ02.02 закрыта": DD7_DI.19, pin 8 "ЗДЭ02.08 открыта": DD7_DI.30, pin 9 "ЗДЭ02.08 закрыта": DD7_DI.31, pin 10 "время движения ЗДЭ": timeToOpenCloseValve, pin 11 "авария питания ЗДЭ02.02": DD9_DI.5, pin 12 "авария питания ЗДЭ02.08": DD9_DI.11)
	(* <- выход использовать в / последнем фильтре для / начала очереди заново *)
	(* если открыт = промывка *)
	(* если открыт = фильтрация *)
	out 1 "следующий в очереди" <= #1060.output
	out 2 "промыть ФС02.01.02" <= #1059
	#1058 ZD0202:SimpleValve(inputOpen: NOT #1059, inputClose: #1059, statusOpen: pin 6, statusClose: pin 7, reset: pin 4, timeToOpenClose: pin 10)
	out 5 "открыть ЗДЭ02.02" <= #1058.outputOpen
	out 6 "закрыть ЗДЭ02.02" <= #1058.outputClose
	out 7 "авария открытия ЗДЭ02.02" <= #1058.errorToOpen
	#1059 OR(panTestValvesFS020102, #1060.regenFilterOUT)
	out 8 "авария закрытия ЗДЭ02.02" <= #1058.errorToClose
	#1060 FS020102manager:FilterQueueManager(input: pin 1, filterAlarm: #1061, regenFilterStatus: pin 3, alarmReset: pin 4, startNextLoop: pin 5)
	#1061 OR(alarmZD020208, pin 2, pin 11, pin 12)
	#1062 OR(#1058.errorToOpen, #1058.errorToClose, #1064.errorToOpen, #1064.errorToClose)
	#1063 alarmZD020208 <= #1062
	out 3 "ФС02.01.02 промыт" <= #1060.regenerated
	out 4 "не удалось промыть" <= #1060.failToRegen
	#1064 ZD0208:SimpleValve(inputOpen: #1059, inputClose: NOT #1059, statusOpen: pin 8, statusClose: pin 9, reset: pin 4, timeToOpenClose: pin 10)
	out 9 "открыть ЗДЭ02.08" <= #1064.outputOpen
	out 10 "закрыть ЗДЭ02.08" <= #1064.outputClose
	out 11 "авария открытия ЗДЭ02.08" <= #1064.errorToOpen
	out 12 "авария закрытия ЗДЭ02.08" <= #1064.errorToClose
END_MACRO
#1065 DD2_DO.5 <= #1057.out 2
#1066 regeneratedFS020102 <= #1057.out 3
#1067 filterFailToRegen020102 <= #1057.out 4
#1068 DD2_DO.18 <= #1057.out 5
#1069 DD2_DO.19 <= #1057.out 6
#1070 errorToOpenZD0202 <= #1057.out 7
#1071 errorToCloseZD0202 <= #1057.out 8
#1072 DD2_DO.30 <= #1057.out 9
#1073 DD2_DO.31 <= #1057.out 10
#1074 errorToOpenZD0208 <= #1057.out 11
#1075 errorToCloseZD0208 <= #1057.out 12
#1076 MACRO управление промывкой фильтра ФС02.01.03(pin 1 "сигнал на промывку": #1057.out 1, pin 2 "авария фильтра": DD6_DI.25, pin 3 "подтверждение промывки": DD6_DI.24, pin 4 "сброс аварий": alarmReset, pin 5 "начать очередь снова": filterStartNewQueue, pin 6 "ЗДЭ02.03 открыта": DD7_DI.20, pin 7 "ЗДЭ02.03 закрыта": DD7_DI.21, pin 8 "ЗДЭ02.09 открыта": DD8_DI.0, pin 9 "ЗДЭ02.09 закрыта": DD8_DI.1, pin 10 "время движения ЗДЭ": timeToOpenCloseValve, pin 11 "авария питания ЗДЭ02.03": DD9_DI.6, pin 12 "авария питания ЗДЭ02.09": DD9_DI.12)
	(* <- выход использовать в / последнем фильтре для / начала очереди заново *)
	(* если открыт = промывка *)
	(* если открыт = фильтрация *)
	out 1 "следующий в очереди" <= #1079.output
	out 2 "промыть ФС02.01.03" <= #1078
	#1077 ZD0203:SimpleValve(inputOpen: NOT #1078, inputClose: #1078, statusOpen: pin 6, statusClose: pin 7, reset: pin 4, timeToOpenClose: pin 10)
	out 5 "открыть ЗДЭ02.03" <= #1077.outputOpen
	out 6 "закрыть ЗДЭ02.03" <= #1077.outputClose
	out 7 "авария открытия ЗДЭ02.03" <= #1077.errorToOpen
	#1078 OR(panTestValvesFS020103, #1079.regenFilterOUT)
	out 8 "авария закрытия ЗДЭ02.03" <= #1077.errorToClose
	#1079 FS020103manager:FilterQueueManager(input: pin 1, filterAlarm: #1080, regenFilterStatus: pin 3, alarmReset: pin 4, startNextLoop: pin 5)
	#1080 OR(alarmZD020309, pin 2, pin 11, pin 12)
	#1081 OR(#1077.errorToOpen, #1077.errorToClose, #1083.errorToOpen, #1083.errorToClose)
	#1082 alarmZD020309 <= #1081
	out 3 "ФС02.01.03 промыт" <= #1079.regenerated
	out 4 "не удалось промыть" <= #1079.failToRegen
	#1083 ZD0209:SimpleValve(inputOpen: #1078, inputClose: NOT #1078, statusOpen: pin 8, statusClose: pin 9, reset: pin 4, timeToOpenClose: pin 10)
	out 9 "открыть ЗДЭ02.09" <= #1083.outputOpen
	out 10 "закрыть ЗДЭ02.09" <= #1083.outputClose
	out 11 "авария открытия ЗДЭ02.09" <= #1083.errorToOpen
	out 12 "авария закрытия ЗДЭ02.09" <= #1083.errorToClose
END_MACRO
#1084 DD2_DO.6 <= #1076.out 2
#1085 regeneratedFS020103 <= #1076.out 3
#1086 filterFailToRegen020103 <= #1076.out 4
#1087 DD2_DO.20 <= #1076.out 5
#1088 DD2_DO.21 <= #1076.out 6
#1089 errorToOpenZD0203 <= #1076.out 7
#1090 errorToCloseZD0203 <= #1076.out 8
#1091 DD3_DO.0 <= #1076.out 9
#1092 DD3_DO.1 <= #1076.out 10
#1093 errorToOpenZD0209 <= #1076.out 11
#1094 errorToCloseZD0209 <= #1076.out 12
#1095 MACRO управление промывкой фильтра ФС02.01.04(pin 1 "сигнал на промывку": #1076.out 1, pin 2 "авария фильтра": DD6_DI.27, pin 3 "подтверждение промывки": DD6_DI.26, pin 4 "сброс аварий": alarmReset, pin 5 "начать очередь снова": filterStartNewQueue, pin 6 "ЗДЭ02.04 открыта": DD7_DI.22, pin 7 "ЗДЭ02.04 закрыта": DD7_DI.23, pin 8 "ЗДЭ02.10 открыта": DD8_DI.2, pin 9 "ЗДЭ02.10 закрыта": DD8_DI.3, pin 10 "время движения ЗДЭ": timeToOpenCloseValve, pin 11 "авария питания ЗДЭ02.04": DD9_DI.7, pin 12 "авария питания ЗДЭ02.10": DD9_DI.13)
	(* <- выход использовать в / последнем фильтре для / начала очереди заново *)
	(* если открыт = промывка *)
	(* если открыт = фильтрация *)
	out 1 "следующий в очереди" <= #1098.output
	out 2 "промыть ФС02.01.04" <= #1097
	#1096 ZD0204:SimpleValve(inputOpen: NOT #1097, inputClose: #1097, statusOpen: pin 6, statusClose: pin 7, reset: pin 4, timeToOpenClose: pin 10)
	out 5 "открыть ЗДЭ02.04" <= #1096.outputOpen
	out 6 "закрыть ЗДЭ02.04" <= #1096.outputClose
	out 7 "авария открытия ЗДЭ02.04" <= #1096.errorToOpen
	#1097 OR(panTestValvesFS020104, #1098.regenFilterOUT)
	out 8 "авария закрытия ЗДЭ02.04" <= #1096.errorToClose
	#1098 FS020104manager:FilterQueueManager(input: pin 1, filterAlarm: #1099, regenFilterStatus: pin 3, alarmReset: pin 4, startNextLoop: pin 5)
	#1099 OR(alarmZD020410, pin 2, pin 11, pin 12)
	#1100 OR(#1096.errorToOpen, #1096.errorToClose, #1102.errorToOpen, #1102.errorToClose)
	#1101 alarmZD020410 <= #1100
	out 3 "ФС02.01.04 промыт" <= #1098.regenerated
	out 4 "не удалось промыть" <= #1098.failToRegen
	#1102 ZD0210:SimpleValve(inputOpen: #1097, inputClose: NOT #1097, statusOpen: pin 8, statusClose: pin 9, reset: pin 4, timeToOpenClose: pin 10)
	out 9 "открыть ЗДЭ02.10" <= #1102.outputOpen
	out 10 "закрыть ЗДЭ02.10" <= #1102.outputClose
	out 11 "авария открытия ЗДЭ02.10" <= #1102.errorToOpen
	out 12 "авария закрытия ЗДЭ02.10" <= #1102.errorToClose
END_MACRO
#1103 DD2_DO.7 <= #1095.out 2
#1104 regeneratedFS020104 <= #1095.out 3
#1105 filterFailToRegen020104 <= #1095.out 4
#1106 DD2_DO.22 <= #1095.out 5
#1107 DD2_DO.23 <= #1095.out 6
#1108 errorToOpenZD0204 <= #1095.out 7
#1109 errorToCloseZD0204 <= #1095.out 8
#1110 DD3_DO.2 <= #1095.out 9
#1111 DD3_DO.3 <= #1095.out 10
#1112 errorToOpenZD0210 <= #1095.out 11
#1113 errorToCloseZD0210 <= #1095.out 12
#1114 MACRO управление промывкой фильтра ФС02.01.05(pin 1 "сигнал на промывку": #1095.out 1, pin 2 "авария фильтра": DD6_DI.29, pin 3 "подтверждение промывки": DD6_DI.28, pin 4 "сброс аварий": alarmReset, pin 5 "начать очередь снова": filterStartNewQueue, pin 6 "ЗДЭ02.05 открыта": DD7_DI.24, pin 7 "ЗДЭ02.05 закрыта": DD7_DI.25, pin 8 "ЗДЭ02.11 открыта": DD8_DI.4, pin 9 "ЗДЭ02.11 закрыта": DD8_DI.5, pin 10 "время движения ЗДЭ": timeToOpenCloseValve, pin 11 "авария питания ЗДЭ02.05": DD9_DI.8, pin 12 "авария питания ЗДЭ02.11": DD9_DI.14)
	(* <- выход использовать в / последнем фильтре для / начала очереди заново *)
	(* если открыт = промывка *)
	(* если открыт = фильтрация *)
	out 1 "следующий в очереди" <= #1117.output
	out 2 "промыть ФС02.01.05" <= #1116
	#1115 ZD0205:SimpleValve(inputOpen: NOT #1116, inputClose: #1116, statusOpen: pin 6, statusClose: pin 7, reset: pin 4, timeToOpenClose: pin 10)
	out 5 "открыть ЗДЭ02.05" <= #1115.outputOpen
	out 6 "закрыть ЗДЭ02.05" <= #1115.outputClose
	out 7 "авария открытия ЗДЭ02.05" <= #1115.errorToOpen
	#1116 OR(panTestValvesFS020105, #1117.regenFilterOUT)
	out 8 "авария закрытия ЗДЭ02.05" <= #1115.errorToClose
	#1117 FS020105manager:FilterQueueManager(input: pin 1, filterAlarm: #1118, regenFilterStatus: pin 3, alarmReset: pin 4, startNextLoop: pin 5)
	#1118 OR(alarmZD020511, pin 2, pin 11, pin 12)
	#1119 OR(#1115.errorToOpen, #1115.errorToClose, #1121.errorToOpen, #1121.errorToClose)
	#1120 alarmZD020511 <= #1119
	out 3 "ФС02.01.05 промыт" <= #1117.regenerated
	out 4 "не удалось промыть" <= #1117.failToRegen
	#1121 ZD0211:SimpleValve(inputOpen: #1116, inputClose: NOT #1116, statusOpen: pin 8, statusClose: pin 9, reset: pin 4, timeToOpenClose: pin 10)
	out 9 "открыть ЗДЭ02.11" <= #1121.outputOpen
	out 10 "закрыть ЗДЭ02.11" <= #1121.outputClose
	out 11 "авария открытия ЗДЭ02.11" <= #1121.errorToOpen
	out 12 "авария закрытия ЗДЭ02.11" <= #1121.errorToClose
END_MACRO
#1122 DD2_DO.8 <= #1114.out 2
#1123 regeneratedFS020105 <= #1114.out 3
#1124 filterFailToRegen020105 <= #1114.out 4
#1125 DD2_DO.24 <= #1114.out 5
#1126 DD2_DO.25 <= #1114.out 6
#1127 errorToOpenZD0205 <= #1114.out 7
#1128 errorToCloseZD0205 <= #1114.out 8
#1129 DD3_DO.4 <= #1114.out 9
#1130 DD3_DO.5 <= #1114.out 10
#1131 errorToOpenZD0211 <= #1114.out 11
#1132 errorToCloseZD0211 <= #1114.out 12
#1133 MACRO управление промывкой фильтра ФС02.01.06(pin 1 "сигнал на промывку": #1114.out 1, pin 2 "авария фильтра": DD6_DI.31, pin 3 "подтверждение промывки": DD6_DI.30, pin 4 "сброс аварий": alarmReset, pin 5 "начать очередь снова": filterStartNewQueue, pin 6 "ЗДЭ02.06 открыта": DD7_DI.26, pin 7 "ЗДЭ02.06 закрыта": DD7_DI.27, pin 8 "ЗДЭ02.12 открыта": DD8_DI.6, pin 9 "ЗДЭ02.12 закрыта": DD8_DI.7, pin 10 "время движения ЗДЭ": timeToOpenCloseValve, pin 11 "авария питания ЗДЭ02.06": DD9_DI.9, pin 12 "авария питания ЗДЭ02.12": DD9_DI.15)
	(* <- выход использовать в / последнем фильтре для / начала очереди заново *)
	(* если открыт = промывка *)
	(* если открыт = фильтрация *)
	out 1 "следующий в очереди" <= #1136.output
	out 2 "промыть ФС02.01.06" <= #1135
	#1134 ZD0206:SimpleValve(inputOpen: NOT #1135, inputClose: #1135, statusOpen: pin 6, statusClose: pin 7, reset: pin 4, timeToOpenClose: pin 10)
	out 5 "открыть ЗДЭ02.06" <= #1134.outputOpen
	out 6 "закрыть ЗДЭ02.06" <= #1134.outputClose
	out 7 "авария открытия ЗДЭ02.06" <= #1134.errorToOpen
	#1135 OR(panTestValvesFS020106, #1136.regenFilterOUT)
	out 8 "авария закрытия ЗДЭ02.06" <= #1134.errorToClose
	#1136 FS020106manager:FilterQueueManager(input: pin 1, filterAlarm: #1137, regenFilterStatus: pin 3, alarmReset: pin 4, startNextLoop: pin 5)
	#1137 OR(alarmZD020612, pin 2, pin 11, pin 12)
	#1138 OR(#1134.errorToOpen, #1134.errorToClose, #1140.errorToOpen, #1140.errorToClose)
	#1139 alarmZD020612 <= #1138
	out 3 "ФС02.01.06 промыт" <= #1136.regenerated
	out 4 "не удалось промыть" <= #1136.failToRegen
	#1140 ZD0212:SimpleValve(inputOpen: #1135, inputClose: NOT #1135, statusOpen: pin 8, statusClose: pin 9, reset: pin 4, timeToOpenClose: pin 10)
	out 9 "открыть ЗДЭ02.12" <= #1140.outputOpen
	out 10 "закрыть ЗДЭ02.12" <= #1140.outputClose
	out 11 "авария открытия ЗДЭ02.12" <= #1140.errorToOpen
	out 12 "авария закрытия ЗДЭ02.12" <= #1140.errorToClose
END_MACRO
#1141 DD2_DO.9 <= #1133.out 2
#1142 regeneratedFS020106 <= #1133.out 3
#1143 filterFailToRegen020106 <= #1133.out 4
#1144 DD2_DO.26 <= #1133.out 5
#1145 DD2_DO.27 <= #1133.out 6
#1146 errorToOpenZD0206 <= #1133.out 7
#1147 errorToCloseZD0206 <= #1133.out 8
#1148 DD3_DO.6 <= #1133.out 9
#1149 DD3_DO.7 <= #1133.out 10
#1150 errorToOpenZD0212 <= #1133.out 11
#1151 errorToCloseZD0212 <= #1133.out 12
#1152 MACRO управление промывкой фильтра ФС02.02.01(pin 1 "сигнал на промывку": #1133.out 1, pin 2 "авария фильтра": DD7_DI.1, pin 3 "подтверждение промывки": DD7_DI.0, pin 4 "сброс аварий": alarmReset, pin 5 "начать очередь снова": filterStartNewQueue, pin 6 "ЗДЭ02.13 открыта": DD8_DI.8, pin 7 "ЗДЭ02.13 закрыта": DD8_DI.9, pin 8 "ЗДЭ02.19 открыта": DD8_DI.20, pin 9 "ЗДЭ02.19 закрыта": DD8_DI.21, pin 10 "время движения ЗДЭ": timeToOpenCloseValve, pin 11 "авария питания ЗДЭ02.13": DD9_DI.16, pin 12 "авария питания ЗДЭ02.19": DD9_DI.22)
	(* <- выход использовать в / последнем фильтре для / начала очереди заново *)
	(* если открыт = промывка *)
	(* если открыт = фильтрация *)
	out 1 "следующий в очереди" <= #1155.output
	out 2 "промыть ФС02.02.01" <= #1154
	#1153 ZD0213:SimpleValve(inputOpen: NOT #1154, inputClose: #1154, statusOpen: pin 6, statusClose: pin 7, reset: pin 4, timeToOpenClose: pin 10)
	out 5 "открыть ЗДЭ02.13" <= #1153.outputOpen
	out 6 "закрыть ЗДЭ02.13" <= #1153.outputClose
